// Functions/Drawing/F_VN_DrawMatchesExp

	{attribute 'TcIecLibraryType'}
	{attribute 'external_name' := 'F_VN_DrawMatchesExp_GUID_C69E0A3C_7312_D2B7_BD5B_52E833304808'}
	(* Draws the keypoints and matches for visualization purpose. (expert function) *)
	FUNCTION F_VN_DrawMatchesExp : HRESULT
	VAR_INPUT
		ipSrcImage1	:	ITcVnImage;	(* Source image 1 (elements of type USINT) *)
		ipKeyPoints1	:	ITcVnContainer;	(* Container with the keypoints 1 (ContainerType_Vector_TcVnKeyPoint) *)
		ipSrcImage2	:	ITcVnImage;	(* Source image 2 (elements of type USINT, must have the same number of channels as ipSrcImage1) *)
		ipKeyPoints2	:	ITcVnContainer;	(* Container with the keypoints 2 (ContainerType_Vector_TcVnKeyPoint) *)
		ipMatches1To2	:	ITcVnContainer;	(* Container with the descriptor matches (ContainerType_Vector_TcVnDMatch) *)
		ipDestImage	:	REFERENCE TO ITcVnImage;	(* Destination image (An appropriate color image will be created if required.) *)
	END_VAR
	VAR_IN_OUT
		aMatchColor	:	TcVnVector4_LREAL;	(* Color to draw the matches (for {-1, -1, -1, -1}, a random color is chosen for each point and line) *)
		aSingleColor	:	TcVnVector4_LREAL;	(* Color to draw the single keypoints (for {-1, -1, -1, -1}, a random color is chosen for each point) *)
	END_VAR
	VAR_INPUT
		ipMatchesMask	:	ITcVnContainer;	(* Mask to select the matches to be drawn (ContainerType_Vector_SINT; Set to 0 if all matches should be drawn.) *)
		eFlags	:	ETcVnDrawMatchesFlags;	(* A combination of flags to support overdrawing an existing destination image and/or drawing additional (Rich-)Keypoint information (size and orientation) and/or skipping single keypoints *)
		hrPrev	:	HRESULT;	(* HRESULT indicating the result of previous operations (If SUCCEEDED(hrPrev) equals false, no operation is executed.) *)
	END_VAR

END_FUNCTION

// Functions/Drawing/F_VN_DrawOrientation

	{attribute 'TcIecLibraryType'}
	{attribute 'external_name' := 'F_VN_DrawOrientation_GUID_8C5CCEF9_05D8_D749_BE94_0462EB58FE1E'}
	(* Draw the main axis of a set of points/contour based on a rotated rectangle. *)
	FUNCTION F_VN_DrawOrientation : HRESULT
	VAR_IN_OUT
		stOrientation	:	TcVnRotatedRectangle;	(* Rotated rectangle, containig center of mass, lenghts of axes, and rotation angle in clockwise direction *)
	END_VAR
	VAR_INPUT
		ipDestImage	:	ITcVnImage;	(* Destination image *)
	END_VAR
	VAR_IN_OUT
		aColorMainAxis	:	TcVnVector4_LREAL;	(* Color of the major axis *)
	END_VAR
	VAR_INPUT
		nThickness	:	DINT;	(* Line thickness *)
		hrPrev	:	HRESULT;	(* HRESULT indicating the result of previous operations (If SUCCEEDED(hrPrev) equals false, no operation is executed.) *)
	END_VAR

END_FUNCTION

// Functions/Drawing/F_VN_DrawOrientationExp

	{attribute 'TcIecLibraryType'}
	{attribute 'external_name' := 'F_VN_DrawOrientationExp_GUID_696CB60D_07A4_DDA6_8A99_EB0492A244F0'}
	(* Draw the main axis, the horizontal axis and the angle of a set of points/contour based on a rotated rectangle. (expert function) *)
	FUNCTION F_VN_DrawOrientationExp : HRESULT
	VAR_IN_OUT
		stOrientation	:	TcVnRotatedRectangle;	(* Rotated rectangle, containig center of mass, lenghts of axes, and rotation angle in clockwise direction *)
	END_VAR
	VAR_INPUT
		ipDestImage	:	ITcVnImage;	(* Destination image *)
	END_VAR
	VAR_IN_OUT
		aColorMainAxis	:	TcVnVector4_LREAL;	(* Color of the major axis *)
	END_VAR
	VAR_INPUT
		nThickness	:	DINT;	(* Line thickness *)
	END_VAR
	VAR_IN_OUT
		aColorHorizontalAxis	:	TcVnVector4_LREAL;	(* Color of the horizontal axis *)
	END_VAR
	VAR_INPUT
		fFontScale	:	LREAL;	(* Scaling factor for the text *)
		hrPrev	:	HRESULT;	(* HRESULT indicating the result of previous operations (If SUCCEEDED(hrPrev) equals false, no operation is executed.) *)
	END_VAR

END_FUNCTION

// Functions/Drawing/F_VN_DrawPoint

	{attribute 'TcIecLibraryType'}
	{attribute 'external_name' := 'F_VN_DrawPoint_GUID_EB197B9A_8498_D424_9F64_30D926D7A450'}
	(* Draws a point. *)
	FUNCTION F_VN_DrawPoint : HRESULT
	VAR_INPUT
		nX	:	UDINT;	(* x coordinate of the point *)
		nY	:	UDINT;	(* y coordinate of the point *)
		ipDestImage	:	ITcVnImage;	(* Destination image *)
		eShape	:	ETcVnDrawShape;	(* Point shape *)
	END_VAR
	VAR_IN_OUT
		aColor	:	TcVnVector4_LREAL;	(* Color (for {-1, -1, -1, -1}, a random color is chosen) *)
	END_VAR
	VAR_INPUT
		hrPrev	:	HRESULT;	(* HRESULT indicating the result of previous operations (If SUCCEEDED(hrPrev) equals false, no operation is executed.) *)
	END_VAR

END_FUNCTION

// Functions/Drawing/F_VN_DrawPointExp

	{attribute 'TcIecLibraryType'}
	{attribute 'external_name' := 'F_VN_DrawPointExp_GUID_0CB1EFC6_EA71_DD9E_A07B_08DD7C0269E3'}
	(* Draw a point. (expert function) *)
	FUNCTION F_VN_DrawPointExp : HRESULT
	VAR_INPUT
		nX	:	UDINT;	(* x coordinate of the point *)
		nY	:	UDINT;	(* y coordinate of the point *)
		ipDestImage	:	ITcVnImage;	(* Destination image *)
		eShape	:	ETcVnDrawShape;	(* Point shape *)
	END_VAR
	VAR_IN_OUT
		aColor	:	TcVnVector4_LREAL;	(* Color (for {-1, -1, -1, -1}, a random color is chosen) *)
	END_VAR
	VAR_INPUT
		nSize	:	UDINT;	(* Size of the shape (half width) *)
		nThickness	:	DINT;	(* Line thickness (if negative, the shape is filled if it is closed) *)
		eLineType	:	ETcVnLineType;	(* Line type *)
		hrPrev	:	HRESULT;	(* HRESULT indicating the result of previous operations (If SUCCEEDED(hrPrev) equals false, no operation is executed.) *)
	END_VAR

END_FUNCTION

// Functions/Drawing/F_VN_DrawPoints

	{attribute 'TcIecLibraryType'}
	{attribute 'external_name' := 'F_VN_DrawPoints_GUID_E6C839DF_E6AE_DD7C_B6D1_DE7AB7EFA551'}
	(* Draw a collection of points. *)
	FUNCTION F_VN_DrawPoints : HRESULT
	VAR_INPUT
		ipPoints	:	ITcVnContainer;	(* Container with TcVnPoint2_DINT or TcVnPoint2_REAL elements *)
		ipDestImage	:	ITcVnImage;	(* Destination image *)
		eShape	:	ETcVnDrawShape;	(* Point shape *)
	END_VAR
	VAR_IN_OUT
		aColor	:	TcVnVector4_LREAL;	(* Color (for {-1, -1, -1, -1}, a random color is chosen for each point) *)
	END_VAR
	VAR_INPUT
		hrPrev	:	HRESULT;	(* HRESULT indicating the result of previous operations (If SUCCEEDED(hrPrev) equals false, no operation is executed.) *)
	END_VAR

END_FUNCTION

// Functions/Drawing/F_VN_DrawPointsExp

	{attribute 'TcIecLibraryType'}
	{attribute 'external_name' := 'F_VN_DrawPointsExp_GUID_34B2960B_E925_DF02_A623_3F9677F5FB98'}
	(* Draw a collection of points. (expert function) *)
	FUNCTION F_VN_DrawPointsExp : HRESULT
	VAR_INPUT
		ipPoints	:	ITcVnContainer;	(* Container with TcVnPoint2_DINT or TcVnPoint2_REAL elements *)
		ipDestImage	:	ITcVnImage;	(* Destination image *)
		eShape	:	ETcVnDrawShape;	(* Point shape *)
	END_VAR
	VAR_IN_OUT
		aColor	:	TcVnVector4_LREAL;	(* Color (for {-1, -1, -1, -1}, a random color is chosen for each point) *)
	END_VAR
	VAR_INPUT
		nSize	:	UDINT;	(* Size of the shape (half width) *)
		nThickness	:	DINT;	(* Line thickness (if negative, the shape is filled if it is closed) *)
		eLineType	:	ETcVnLineType;	(* Line type *)
		hrPrev	:	HRESULT;	(* HRESULT indicating the result of previous operations (If SUCCEEDED(hrPrev) equals false, no operation is executed.) *)
	END_VAR

END_FUNCTION

// Functions/Drawing/F_VN_DrawPolygon

	{attribute 'TcIecLibraryType'}
	{attribute 'external_name' := 'F_VN_DrawPolygon_GUID_2AC3D600_E474_DEFB_A3DB_E972A97945F6'}
	(* Draw a pologon using collection of points. *)
	FUNCTION F_VN_DrawPolygon : HRESULT
	VAR_INPUT
		ipPoints	:	ITcVnContainer;	(* Container with TcVnPoint2_DINT, TcVnPoint2_REAL, or TcVnPoint2_LREAL elements *)
		ipDestImage	:	ITcVnImage;	(* Destination image *)
	END_VAR
	VAR_IN_OUT
		aColor	:	TcVnVector4_LREAL;	(* Color *)
	END_VAR
	VAR_INPUT
		nThickness	:	DINT;	(* Line thickness (if negative, the polygon is filled) *)
		hrPrev	:	HRESULT;	(* HRESULT indicating the result of previous operations (If SUCCEEDED(hrPrev) equals false, no operation is executed.) *)
	END_VAR

END_FUNCTION

// Functions/Drawing/F_VN_DrawPolygonExp

	{attribute 'TcIecLibraryType'}
	{attribute 'external_name' := 'F_VN_DrawPolygonExp_GUID_D79A9437_66CC_D2F2_AC2B_AABA5EDF4A83'}
	(* Draw a pologon using collection of points. (expert function) *)
	FUNCTION F_VN_DrawPolygonExp : HRESULT
	VAR_INPUT
		ipPoints	:	ITcVnContainer;	(* Container with TcVnPoint2_DINT, TcVnPoint2_REAL, or TcVnPoint2_LREAL elements *)
		ipDestImage	:	ITcVnImage;	(* Destination image *)
	END_VAR
	VAR_IN_OUT
		aColor	:	TcVnVector4_LREAL;	(* Color *)
	END_VAR
	VAR_INPUT
		nThickness	:	DINT;	(* Line thickness (if negative, the shape is filled) *)
		bIsClosed	:	BOOL;	(* If it is true, the function draws a line from the last point to the first point to close the polygon. *)
		eLineType	:	ETcVnLineType;	(* Line type *)
		nShift	:	UDINT;	(* Fractional bits of the coordinates (bit shift) *)
		hrPrev	:	HRESULT;	(* HRESULT indicating the result of previous operations (If SUCCEEDED(hrPrev) equals false, no operation is executed.) *)
	END_VAR

END_FUNCTION

// Functions/Drawing/F_VN_DrawRectangle

	{attribute 'TcIecLibraryType'}
	{attribute 'external_name' := 'F_VN_DrawRectangle_GUID_CA7621FD_AAA8_DD79_BAA6_54BF18EEF247'}
	(* Draw a rectangle. *)
	FUNCTION F_VN_DrawRectangle : HRESULT
	VAR_INPUT
		nTopLeftX	:	UDINT;	(* x coordinate of the top left corner *)
		nTopLeftY	:	UDINT;	(* y coordinate of the top left corner *)
		nBottomRightX	:	UDINT;	(* x coordinate of the bottom right corner *)
		nBottomRightY	:	UDINT;	(* y coordinate of the bottom right corner *)
		ipDestImage	:	ITcVnImage;	(* Destination image *)
	END_VAR
	VAR_IN_OUT
		aColor	:	TcVnVector4_LREAL;	(* Color *)
	END_VAR
	VAR_INPUT
		nThickness	:	DINT;	(* Line thickness (if negative, the rectangle is filled) *)
		hrPrev	:	HRESULT;	(* HRESULT indicating the result of previous operations (If SUCCEEDED(hrPrev) equals false, no operation is executed.) *)
	END_VAR

END_FUNCTION

// Functions/Drawing/F_VN_DrawRectangle_TcVnRectangle_DINT

	{attribute 'TcIecLibraryType'}
	{attribute 'external_name' := 'F_VN_DrawRectangle_TcVnRectangle_DINT_GUID_35950137_42A1_DD6B_8040_5531524BF69E'}
	(* Draw a rectangle. *)
	FUNCTION F_VN_DrawRectangle_TcVnRectangle_DINT : HRESULT
	VAR_IN_OUT
		stRectangle	:	TcVnRectangle_DINT;	(* Rectangle to be drawn *)
	END_VAR
	VAR_INPUT
		ipDestImage	:	ITcVnImage;	(* Destination image *)
	END_VAR
	VAR_IN_OUT
		aColor	:	TcVnVector4_LREAL;	(* Color *)
	END_VAR
	VAR_INPUT
		nThickness	:	DINT;	(* Line thickness (if negative, the rectangle is filled) *)
		hrPrev	:	HRESULT;	(* HRESULT indicating the result of previous operations (If SUCCEEDED(hrPrev) equals false, no operation is executed.) *)
	END_VAR

END_FUNCTION

// Functions/Drawing/F_VN_DrawRectangle_TcVnRectangle_UDINT

	{attribute 'TcIecLibraryType'}
	{attribute 'external_name' := 'F_VN_DrawRectangle_TcVnRectangle_UDINT_GUID_4B7204C8_DED8_DFCB_8469_BEF3FFA8576B'}
	(* Draw a rectangle. *)
	FUNCTION F_VN_DrawRectangle_TcVnRectangle_UDINT : HRESULT
	VAR_IN_OUT
		stRectangle	:	TcVnRectangle_UDINT;	(* Rectangle to be drawn *)
	END_VAR
	VAR_INPUT
		ipDestImage	:	ITcVnImage;	(* Destination image *)
	END_VAR
	VAR_IN_OUT
		aColor	:	TcVnVector4_LREAL;	(* Color *)
	END_VAR
	VAR_INPUT
		nThickness	:	DINT;	(* Line thickness (if negative, the rectangle is filled) *)
		hrPrev	:	HRESULT;	(* HRESULT indicating the result of previous operations (If SUCCEEDED(hrPrev) equals false, no operation is executed.) *)
	END_VAR

END_FUNCTION

// Functions/Drawing/F_VN_DrawRotatedRectangle

	{attribute 'TcIecLibraryType'}
	{attribute 'external_name' := 'F_VN_DrawRotatedRectangle_GUID_E91FE6CA_6FE6_D9DD_B4B2_DB4AEAF725E4'}
	(* Draw a rectangle. *)
	FUNCTION F_VN_DrawRotatedRectangle : HRESULT
	VAR_IN_OUT
		stRectangle	:	TcVnRotatedRectangle;	(* Rectangle to be drawn (rotation angle in degrees) *)
	END_VAR
	VAR_INPUT
		ipDestImage	:	ITcVnImage;	(* Destination image *)
	END_VAR
	VAR_IN_OUT
		aColor	:	TcVnVector4_LREAL;	(* Color *)
	END_VAR
	VAR_INPUT
		nThickness	:	DINT;	(* Line thickness (if negative, the rectangle is filled) *)
		hrPrev	:	HRESULT;	(* HRESULT indicating the result of previous operations (If SUCCEEDED(hrPrev) equals false, no operation is executed.) *)
	END_VAR

END_FUNCTION

// Functions/Drawing/F_VN_DrawRotatedRectangleExp

	{attribute 'TcIecLibraryType'}
	{attribute 'external_name' := 'F_VN_DrawRotatedRectangleExp_GUID_FE06CB4F_97F7_D420_BF0D_F8C392244530'}
	(* Draw a rectangle. (expert function) *)
	FUNCTION F_VN_DrawRotatedRectangleExp : HRESULT
	VAR_IN_OUT
		stRectangle	:	TcVnRotatedRectangle;	(* Rectangle to be drawn (rotation angle in degrees) *)
	END_VAR
	VAR_INPUT
		ipDestImage	:	ITcVnImage;	(* Destination image *)
	END_VAR
	VAR_IN_OUT
		aColor	:	TcVnVector4_LREAL;	(* Color *)
	END_VAR
	VAR_INPUT
		nThickness	:	DINT;	(* Line thickness (if negative, the rectangle is filled) *)
		eLineType	:	ETcVnLineType;	(* Line type *)
		hrPrev	:	HRESULT;	(* HRESULT indicating the result of previous operations (If SUCCEEDED(hrPrev) equals false, no operation is executed.) *)
	END_VAR

END_FUNCTION

// Functions/Drawing/F_VN_FillCircle

	{attribute 'TcIecLibraryType'}
	{attribute 'external_name' := 'F_VN_FillCircle_GUID_57F72791_EAC2_DD4D_87CB_053D8258EE82'}
	(* Paint a filled circle. *)
	FUNCTION F_VN_FillCircle : HRESULT
	VAR_INPUT
		nCenterX	:	UDINT;	(* x coordinate of the center *)
		nCenterY	:	UDINT;	(* y coordinate of the center *)
		nRadius	:	UDINT;	(* Radius *)
		ipDestImage	:	ITcVnImage;	(* Destination image *)
	END_VAR
	VAR_IN_OUT
		aColor	:	TcVnVector4_LREAL;	(* Color *)
	END_VAR
	VAR_INPUT
		hrPrev	:	HRESULT;	(* HRESULT indicating the result of previous operations (If SUCCEEDED(hrPrev) equals false, no operation is executed.) *)
	END_VAR

END_FUNCTION

// Functions/Drawing/F_VN_FillContours

	{attribute 'TcIecLibraryType'}
	{attribute 'external_name' := 'F_VN_FillContours_GUID_9A17D4B9_08AB_D368_B51D_AE757CA4E5B1'}
	(* Paint a single point set or multiple point sets that are interpreted as contours. *)
	FUNCTION F_VN_FillContours : HRESULT
	VAR_INPUT
		ipContours	:	ITcVnContainer;	(* Single contour (ContainerType_Vector_TcVnPoint2_DINT) or multiple contours (ContainerType_Vector_Vector_TcVnPoint2_DINT) *)
		nContourIndex	:	DINT;	(* Index of a specific contour to be drawn (if negative, all contours within the container are drawn) *)
		ipDestImage	:	ITcVnImage;	(* Destination image *)
	END_VAR
	VAR_IN_OUT
		aColor	:	TcVnVector4_LREAL;	(* Color *)
	END_VAR
	VAR_INPUT
		hrPrev	:	HRESULT;	(* HRESULT indicating the result of previous operations (If SUCCEEDED(hrPrev) equals false, no operation is executed.) *)
	END_VAR

END_FUNCTION

// Functions/Drawing/F_VN_FillEllipse

	{attribute 'TcIecLibraryType'}
	{attribute 'external_name' := 'F_VN_FillEllipse_GUID_5CD99C65_85B9_D8C2_BE64_A5A4252AB0BB'}
	(* Paint a filled ellipse. *)
	FUNCTION F_VN_FillEllipse : HRESULT
	VAR_IN_OUT
		stEllipse	:	TcVnRotatedRectangle;	(* Ellipse to be painted (rotation angle in degrees) *)
	END_VAR
	VAR_INPUT
		ipDestImage	:	ITcVnImage;	(* Destination image *)
	END_VAR
	VAR_IN_OUT
		aColor	:	TcVnVector4_LREAL;	(* Color *)
	END_VAR
	VAR_INPUT
		hrPrev	:	HRESULT;	(* HRESULT indicating the result of previous operations (If SUCCEEDED(hrPrev) equals false, no operation is executed.) *)
	END_VAR

END_FUNCTION

// Functions/Drawing/F_VN_FillPolygon

	{attribute 'TcIecLibraryType'}
	{attribute 'external_name' := 'F_VN_FillPolygon_GUID_25CBE1F6_0702_D828_A491_380DC4B9D8A2'}
	(* Paint a filled pologon using a set of points. *)
	FUNCTION F_VN_FillPolygon : HRESULT
	VAR_INPUT
		ipPoints	:	ITcVnContainer;	(* Container with TcVnPoint2_DINT, TcVnPoint2_REAL, or TcVnPoint2_LREAL elements *)
		ipDestImage	:	ITcVnImage;	(* Destination image *)
	END_VAR
	VAR_IN_OUT
		aColor	:	TcVnVector4_LREAL;	(* Color *)
	END_VAR
	VAR_INPUT
		hrPrev	:	HRESULT;	(* HRESULT indicating the result of previous operations (If SUCCEEDED(hrPrev) equals false, no operation is executed.) *)
	END_VAR

END_FUNCTION

// Functions/Drawing/F_VN_FillRectangle

	{attribute 'TcIecLibraryType'}
	{attribute 'external_name' := 'F_VN_FillRectangle_GUID_B6F6404B_5305_DD2F_82D7_B60633C88882'}
	(* Paint a filled rectangle. *)
	FUNCTION F_VN_FillRectangle : HRESULT
	VAR_INPUT
		nTopLeftX	:	UDINT;	(* x coordinate of the top left corner *)
		nTopLeftY	:	UDINT;	(* y coordinate of the top left corner *)
		nBottomRightX	:	UDINT;	(* x coordinate of the bottom right corner *)
		nBottomRightY	:	UDINT;	(* y coordinate of the bottom right corner *)
		ipDestImage	:	ITcVnImage;	(* Destination image *)
	END_VAR
	VAR_IN_OUT
		aColor	:	TcVnVector4_LREAL;	(* Color *)
	END_VAR
	VAR_INPUT
		hrPrev	:	HRESULT;	(* HRESULT indicating the result of previous operations (If SUCCEEDED(hrPrev) equals false, no operation is executed.) *)
	END_VAR

END_FUNCTION

// Functions/Drawing/F_VN_FillRotatedRectangle

	{attribute 'TcIecLibraryType'}
	{attribute 'external_name' := 'F_VN_FillRotatedRectangle_GUID_051B9FAB_5B48_DFCC_BEE4_115436A91595'}
	(* Paint a filled rectangle. *)
	FUNCTION F_VN_FillRotatedRectangle : HRESULT
	VAR_IN_OUT
		stRectangle	:	TcVnRotatedRectangle;	(* Rectangle to be painted (rotation angle in degrees) *)
	END_VAR
	VAR_INPUT
		ipDestImage	:	ITcVnImage;	(* Destination image *)
	END_VAR
	VAR_IN_OUT
		aColor	:	TcVnVector4_LREAL;	(* Color *)
	END_VAR
	VAR_INPUT
		hrPrev	:	HRESULT;	(* HRESULT indicating the result of previous operations (If SUCCEEDED(hrPrev) equals false, no operation is executed.) *)
	END_VAR

END_FUNCTION

// Functions/Drawing/F_VN_PlotIntensityProfile

	{attribute 'TcIecLibraryType'}
	{attribute 'external_name' := 'F_VN_PlotIntensityProfile_GUID_B2A04906_DDBE_D38C_A697_F571DC74A928'}
	(* Plots the pixel intensity profile along a line segment in an image. *)
	FUNCTION F_VN_PlotIntensityProfile : HRESULT
	VAR_INPUT
		ipSrcImage	:	ITcVnImage;	(* Source image (USINT, 1 channel) *)
		ipDestImage	:	REFERENCE TO ITcVnImage;	(* Destination image (USINT, 1 channel. x: position, y: intensity, origin: bottom left. An appropriate destination image will be created if required.) *)
	END_VAR
	VAR_IN_OUT
		aStartPoint	:	TcVnPoint2_REAL;	(* Start point of the line segment *)
		aEndPoint	:	TcVnPoint2_REAL;	(* End point of the line segment *)
	END_VAR
	VAR_INPUT
		hrPrev	:	HRESULT;	(* HRESULT indicating the result of previous operations (If SUCCEEDED(hrPrev) equals false, no operation is executed.) *)
	END_VAR

END_FUNCTION

// Functions/Drawing/F_VN_PlotIntensityProfileExp

	{attribute 'TcIecLibraryType'}
	{attribute 'external_name' := 'F_VN_PlotIntensityProfileExp_GUID_18DC275F_A530_D420_B515_3BF70FC6163A'}
	(* Plots the pixel intensity profile along a line segment in an image. (expert function) *)
	FUNCTION F_VN_PlotIntensityProfileExp : HRESULT
	VAR_INPUT
		ipSrcImage	:	ITcVnImage;	(* Source image (USINT, 1 channel) *)
		ipDestImage	:	REFERENCE TO ITcVnImage;	(* Destination image (USINT, 1 channel. x: position, y: intensity, origin: bottom left. An appropriate destination image will be created if required.) *)
	END_VAR
	VAR_IN_OUT
		aStartPoint	:	TcVnPoint2_REAL;	(* Start point of the line segment *)
		aEndPoint	:	TcVnPoint2_REAL;	(* End point of the line segment *)
		aBackgroundColor	:	TcVnVector4_LREAL;	(* Background color *)
		aLineColor	:	TcVnVector4_LREAL;	(* Line color *)
		aGridColor	:	TcVnVector4_LREAL;	(* Grid color *)
	END_VAR
	VAR_INPUT
		nScaleX	:	DINT;	(* Scale in x direction (ipDestImage will have a width of nScaleX * (ipSrcImage width - 1) + 1) *)
		nScaleY	:	DINT;	(* Scale in y direction (ipDestImage will have a height of nScaleY * 255 + 1) *)
		nThickness	:	DINT;	(* Line thickness *)
		nDestChannels	:	DINT;	(* ipDestImage channels (1 or 3) *)
		hrPrev	:	HRESULT;	(* HRESULT indicating the result of previous operations (If SUCCEEDED(hrPrev) equals false, no operation is executed.) *)
	END_VAR

END_FUNCTION

// Functions/Drawing/F_VN_PutLabel

	{attribute 'TcIecLibraryType'}
	{attribute 'external_name' := 'F_VN_PutLabel_GUID_AC21311A_53C7_DC28_BB97_DE22D5467497'}
	(* Write a label (black text on white background) into an image. *)
	FUNCTION F_VN_PutLabel : HRESULT
	VAR_IN_OUT CONSTANT
		sText	:	STRING;	(* Text *)
	END_VAR
	VAR_INPUT
		ipDestImage	:	ITcVnImage;	(* Destination image *)
		nX	:	UDINT;	(* x coordinate (bottom left) *)
		nY	:	UDINT;	(* y coordinate (bottom left) *)
		fFontScale	:	LREAL;	(* Scaling factor *)
		hrPrev	:	HRESULT;	(* HRESULT indicating the result of previous operations (If SUCCEEDED(hrPrev) equals false, no operation is executed.) *)
	END_VAR

END_FUNCTION

// Functions/Drawing/F_VN_PutLabelExp

	{attribute 'TcIecLibraryType'}
	{attribute 'external_name' := 'F_VN_PutLabelExp_GUID_22D551B9_953C_DDA8_9D1A_8B55704272D4'}
	(* Write a label (text on unified background) into an image. (expert function) *)
	FUNCTION F_VN_PutLabelExp : HRESULT
	VAR_IN_OUT CONSTANT
		sText	:	STRING;	(* Text *)
	END_VAR
	VAR_INPUT
		ipDestImage	:	ITcVnImage;	(* Destination image *)
		nX	:	UDINT;	(* x coordinate (bottom left) *)
		nY	:	UDINT;	(* y coordinate (bottom left) *)
		fFontScale	:	LREAL;	(* Scaling factor *)
		nThickness	:	UDINT;	(* Line thickness *)
		eFontType	:	ETcVnFontType;	(* Font type *)
	END_VAR
	VAR_IN_OUT
		aFontColor	:	TcVnVector4_LREAL;	(* Font color *)
		aBackgroundColor	:	TcVnVector4_LREAL;	(* Background color *)
	END_VAR
	VAR_INPUT
		eLineType	:	ETcVnLineType;	(* Line type *)
		hrPrev	:	HRESULT;	(* HRESULT indicating the result of previous operations (If SUCCEEDED(hrPrev) equals false, no operation is executed.) *)
	END_VAR

END_FUNCTION

// Functions/Drawing/F_VN_PutText

	{attribute 'TcIecLibraryType'}
	{attribute 'external_name' := 'F_VN_PutText_GUID_8A847AF0_9C61_D376_BA49_31E7BD216F97'}
	(* Write text into an image. *)
	FUNCTION F_VN_PutText : HRESULT
	VAR_IN_OUT CONSTANT
		sText	:	STRING;	(* Text *)
	END_VAR
	VAR_INPUT
		ipDestImage	:	ITcVnImage;	(* Destination image *)
		nX	:	UDINT;	(* x coordinate (bottom left) *)
		nY	:	UDINT;	(* y coordinate (bottom left) *)
		eFontType	:	ETcVnFontType;	(* Font type *)
		fFontScale	:	LREAL;	(* Scaling factor *)
	END_VAR
	VAR_IN_OUT
		aColor	:	TcVnVector4_LREAL;	(* Text color *)
	END_VAR
	VAR_INPUT
		hrPrev	:	HRESULT;	(* HRESULT indicating the result of previous operations (If SUCCEEDED(hrPrev) equals false, no operation is executed.) *)
	END_VAR

END_FUNCTION

// Functions/Drawing/F_VN_PutTextExp

	{attribute 'TcIecLibraryType'}
	{attribute 'external_name' := 'F_VN_PutTextExp_GUID_D88D1077_FEC3_DDA1_8623_3D379A0CC9BD'}
	(* Write text into an image. (expert function) *)
	FUNCTION F_VN_PutTextExp : HRESULT
	VAR_IN_OUT CONSTANT
		sText	:	STRING;	(* Text *)
	END_VAR
	VAR_INPUT
		ipDestImage	:	ITcVnImage;	(* Destination image *)
		nX	:	UDINT;	(* x coordinate (bottom left) *)
		nY	:	UDINT;	(* y coordinate (bottom left) *)
		eFontType	:	ETcVnFontType;	(* Font type *)
		fFontScale	:	LREAL;	(* Scaling factor *)
	END_VAR
	VAR_IN_OUT
		aColor	:	TcVnVector4_LREAL;	(* Text color *)
	END_VAR
	VAR_INPUT
		nThickness	:	DINT;	(* Line thickness *)
		eLineType	:	ETcVnLineType;	(* Line type *)
		bBottomLeftOrigin	:	BOOL;	(* Sets the image origin to the bottom left corner, if true *)
		hrPrev	:	HRESULT;	(* HRESULT indicating the result of previous operations (If SUCCEEDED(hrPrev) equals false, no operation is executed.) *)
	END_VAR

END_FUNCTION

// Functions/Neural Network/F_VN_ConvertDataLayout

	{attribute 'TcIecLibraryType'}
	{attribute 'external_name' := 'F_VN_ConvertDataLayout_GUID_3995A5A2_8722_D5EC_8314_ABF1AA7937E5'}
	(* Convert a data layout (the arrangement of dimensions in the input data) to another data layout. *)
	FUNCTION F_VN_ConvertDataLayout : HRESULT
	VAR_INPUT
		ipSrcImage	:	ITcVnImage;	(* Source image *)
		ipDestImage	:	REFERENCE TO ITcVnImage;	(* Destination image (An appropriate destination image will be created if required.) *)
		nSrcDataLayout	:	ULINT;	(* Data layout of the source image (Commonly used data layouts are available in the enumeration ETcVnDataLayout. If nSrcDataLayout is set to 0 or TCVN_DL_DEFAULT, the DataLayout will be automatically determined based on the dimension of the ipSrcImage: 0x12 for 2D, 0x123 for 3D, 0x1234 for 4D, and so forth.) *)
		nDestDataLayout	:	ULINT;	(* Required output data layout (Commonly used data layouts are available in the enumeration ETcVnDataLayout. nDestDataLayout must not equal 0 or TCVN_DL_DEFAULT.) *)
		hrPrev	:	HRESULT;	(* HRESULT indicating the result of previous operations (If SUCCEEDED(hrPrev) equals false, no operation is executed.) *)
	END_VAR

END_FUNCTION

// Functions/Neural Network/F_VN_ReshapeImage

	{attribute 'TcIecLibraryType'}
	{attribute 'external_name' := 'F_VN_ReshapeImage_GUID_2BBA238A_D9C8_DF6C_A475_21C0DD3F001A'}
	(* Changes the shape of an ITcVnImage. The total number of elements in the new shape must be equal to the total number of elements in ipSrcImage. *)
	FUNCTION F_VN_ReshapeImage : HRESULT
	VAR_INPUT
		ipSrcImage	:	ITcVnImage;	(* Source image (1 channel) *)
		ipDestImage	:	REFERENCE TO ITcVnImage;	(* Destination image (An appropriate single channel destination image will be created if required.) *)
	END_VAR
	VAR_IN_OUT
		aNewShape	:	TcVnArray33_UDINT;	(* Specifies the shape of ipDestImage. First entry is the number of dimensions (max. 32), followed by the sizes of each dimension. If one dimension is set to zero, its value will be automatically calculated based on the total elements of ipSrcImage (Only one dimension can be set to zero.) *)
	END_VAR
	VAR_INPUT
		hrPrev	:	HRESULT;	(* HRESULT indicating the result of previous operations (If SUCCEEDED(hrPrev) equals false, no operation is executed.) *)
	END_VAR

END_FUNCTION

// Functions/Neural Network/F_VN_Sigmoid

	{attribute 'TcIecLibraryType'}
	{attribute 'external_name' := 'F_VN_Sigmoid_GUID_443EE66B_FF0F_D007_AC8F_462BC3F1F276'}
	(* Apply the standard logistic function 1 / (1 + exp(-x)) element-wise to a single- or multi-channel REAL image. *)
	FUNCTION F_VN_Sigmoid : HRESULT
	VAR_INPUT
		ipSrcImage	:	ITcVnImage;	(* Source image (REAL) *)
		ipDestImage	:	REFERENCE TO ITcVnImage;	(* Destination image (An appropriate destination image will be created if required.) *)
		hrPrev	:	HRESULT;	(* HRESULT indicating the result of previous operations (If SUCCEEDED(hrPrev) equals false, no operation is executed.) *)
	END_VAR

END_FUNCTION

// Functions/Neural Network/F_VN_SigmoidExp

	{attribute 'TcIecLibraryType'}
	{attribute 'external_name' := 'F_VN_SigmoidExp_GUID_B65ACE1F_A3FF_DF19_9C9E_6A823D2620ED'}
	(* Apply the logistic function 1 / (1 + exp(-fSteepness * (x - fShift))) element-wise to a single- or multi-channel REAL image. (expert function) *)
	FUNCTION F_VN_SigmoidExp : HRESULT
	VAR_INPUT
		ipSrcImage	:	ITcVnImage;	(* Source image (REAL) *)
		ipDestImage	:	REFERENCE TO ITcVnImage;	(* Destination image (An appropriate destination image will be created if required.) *)
		fShift	:	REAL;	(* Determines the intensity level around which the logistic function transitions. *)
		fSteepness	:	REAL;	(* Controls the sharpness of the transition. *)
		hrPrev	:	HRESULT;	(* HRESULT indicating the result of previous operations (If SUCCEEDED(hrPrev) equals false, no operation is executed.) *)
	END_VAR

END_FUNCTION

// Functions/Neural Network/F_VN_SoftMax

	{attribute 'TcIecLibraryType'}
	{attribute 'external_name' := 'F_VN_SoftMax_GUID_62A1500E_9919_D189_8BB6_E8BC05C5CB3D'}
	(* Apply softmax function pixel-wise to a single channel REAL image. *)
	FUNCTION F_VN_SoftMax : HRESULT
	VAR_INPUT
		ipSrcImage	:	ITcVnImage;	(* Source image (REAL, 1 channel) *)
		ipDestImage	:	REFERENCE TO ITcVnImage;	(* Destination image (An appropriate single channel destination image will be created if required.) *)
		bFlatten	:	BOOL;	(* If true, the resulting image will be reshaped into a single row. *)
		hrPrev	:	HRESULT;	(* HRESULT indicating the result of previous operations (If SUCCEEDED(hrPrev) equals false, no operation is executed.) *)
	END_VAR

END_FUNCTION

// Functions/Neural Network/F_VN_NonMaxSuppression

	{attribute 'TcIecLibraryType'}
	{attribute 'external_name' := 'F_VN_NonMaxSuppression_GUID_DDD612EA_2DB6_D0A1_AA79_316039076A43'}
	(* Perform non-maximum suppression on given bounding boxes and corresponding scores. *)
	FUNCTION F_VN_NonMaxSuppression : HRESULT
	VAR_INPUT
		ipBoundingBoxes	:	ITcVnContainer;	(* Container of bounding boxes to apply the non maximum supresion (ContainerType_Vector_TcVnRectangle_DINT) *)
		ipScores	:	ITcVnContainer;	(* Container of coreeponding score for each bounding box (ContainerType_Vector_REAL) *)
		ipDestIndcies	:	REFERENCE TO ITcVnContainer;	(* Container of the kept indcies after apply the non maximum suppression (ContainerType_Vector_DINT) *)
		fScoreThreshold	:	REAL;	(* A threshold [0.0 to 1.0] used to filter the bounding boxes by score *)
		fOverlapThreshold	:	REAL;	(* A threshold [0.0 to 1.0] that determines the minimum degree of intersection over union (IoU) required for bounding boxes to be considered overlapping *)
		hrPrev	:	HRESULT;	(* HRESULT indicating the result of previous operations (If SUCCEEDED(hrPrev) equals false, no operation is executed.) *)
	END_VAR

END_FUNCTION

// Functions/Neural Network/F_VN_NonMaxSuppressionExp

	{attribute 'TcIecLibraryType'}
	{attribute 'external_name' := 'F_VN_NonMaxSuppressionExp_GUID_254301EF_EB55_D9F0_8663_C0A211C69477'}
	(* Perform non-maximum suppression on given bounding boxes and corresponding scores. (expert function) *)
	FUNCTION F_VN_NonMaxSuppressionExp : HRESULT
	VAR_INPUT
		ipBoundingBoxes	:	ITcVnContainer;	(* Container of bounding boxes to apply the non maximum supresion (ContainerType_Vector_TcVnRectangle_DINT) *)
		ipScores	:	ITcVnContainer;	(* Container of coreeponding score for each bounding box (ContainerType_Vector_REAL) *)
		ipDestIndcies	:	REFERENCE TO ITcVnContainer;	(* Container of the kept indcies after apply the non maximum suppression (ContainerType_Vector_DINT) *)
		fScoreThreshold	:	REAL;	(* A threshold [0.0 to 1.0] used to filter the bounding boxes by score *)
		fOverlapThreshold	:	REAL;	(* A threshold [0.0 to 1.0] that determines the minimum degree of intersection over union (IoU) required for bounding boxes to be considered overlapping *)
		ipClassIndcies	:	ITcVnContainer;	(* Container of corresponding set of class indcies (ContainerType_Vector_DINT) *)
		fEta	:	REAL;	(* An adjustable threshold [0.0 to 1.0] used to dynamically reduce the overlap threshold during processing. Setting it to 1 maintains a constant value for the overlap threshold *)
		nTopK	:	DINT;	(* The maximum number of bounding boxes with the highest scores to undergo the suppression algorithm (must be >= 0). Setting it to zero applies the algorithm to all bounding boxes *)
		hrPrev	:	HRESULT;	(* HRESULT indicating the result of previous operations (If SUCCEEDED(hrPrev) equals false, no operation is executed.) *)
	END_VAR

END_FUNCTION

// Functions/Neural Network/F_VN_ExecuteNeuralNetwork

	{attribute 'TcIecLibraryType'}
	{attribute 'external_name' := 'F_VN_ExecuteNeuralNetwork_GUID_617005B4_6D6B_DC13_A8ED_07F2C339BFC4'}
	(* Execute a neural network using the provided image as input and provide the output of one output layer. The function doesn't perform any pre-processing or transformation. *)
	FUNCTION F_VN_ExecuteNeuralNetwork : HRESULT
	VAR_INPUT
		ipNeuralNetwork	:	ITcVnNeuralNetwork;	(* Neural network model *)
		ipSrcImage	:	ITcVnImage;	(* Source image (The image layout must be adapted to match the model's expected input format using e.g. F_VN_ConvertDataLayout or F_VN_ReshapeImage functions if necessary.) *)
		ipDestImage	:	REFERENCE TO ITcVnImage;	(* Destination image (An appropriate destination image based on the output layer is created. To process the destination image, use e.g. F_VN_ConvertDataLayout or F_VN_ReshapeImage if necessary. *)
		hrPrev	:	HRESULT;	(* HRESULT indicating the result of previous operations (If SUCCEEDED(hrPrev) equals false, no operation is executed.) *)
	END_VAR

END_FUNCTION

// Functions/Neural Network/F_VN_ExecuteNeuralNetwork_MI

	{attribute 'TcIecLibraryType'}
	{attribute 'external_name' := 'F_VN_ExecuteNeuralNetwork_MI_GUID_B9E22B87_BE93_D412_867E_51918F035B7B'}
	(* Execute a neural network with multiple inputs (MI) using the provided images. Ensure all model input names are listed in sInputNames and that the images and names are in the same order. The result of one output layer is returned. The function doesn't perform any pre-processing or transformation. *)
	FUNCTION F_VN_ExecuteNeuralNetwork_MI : HRESULT
	VAR_INPUT
		ipNeuralNetwork	:	ITcVnNeuralNetwork;	(* Neural network model *)
		pSrcImages	:	PVOID;	(* Pointer to an array of source input images *)
		nSrcArraySize	:	UINT;	(* The size of the array referenced by pSrcImages. pSrcImages must reference an array with a size equal to the number of model inputs. *)
	END_VAR
	VAR_IN_OUT CONSTANT
		sInputNames	:	STRING;	(* Input names separated by ";" *)
	END_VAR
	VAR_INPUT
		ipDestImage	:	REFERENCE TO ITcVnImage;	(* Destination image (An appropriate destination image based on the output layer is created. To process the destination image, use e.g. F_VN_ConvertDataLayout or F_VN_ReshapeImage if necessary. *)
		hrPrev	:	HRESULT;	(* HRESULT indicating the result of previous operations (If SUCCEEDED(hrPrev) equals false, no operation is executed.) *)
	END_VAR

END_FUNCTION

// Functions/Neural Network/F_VN_ExecuteNeuralNetwork_MultiLayerOutput

	{attribute 'TcIecLibraryType'}
	{attribute 'external_name' := 'F_VN_ExecuteNeuralNetwork_MultiLayerOutput_GUID_C5CF9BE3_85FE_D822_8CCE_67AE7CEBB5FD'}
	(* This function is deprecated, please use F_VN_ExecuteNeuralNetwork_MO. Execute a neural network using the provided image as input and provide the output of the specified output layers. The function doesn't perform any pre-processing or transformation. *)
	FUNCTION F_VN_ExecuteNeuralNetwork_MultiLayerOutput : HRESULT
	VAR_INPUT
		ipNeuralNetwork	:	ITcVnNeuralNetwork;	(* Neural network model *)
		ipSrcImage	:	ITcVnImage;	(* Source image (The image layout must be adapted to match the model's expected input format using e.g. F_VN_ConvertDataLayout or F_VN_ReshapeImage functions if necessary.) *)
		ipDestImages	:	REFERENCE TO ITcVnContainer;	(* Container of images containing the output from the specified layers. *)
		ipLayerNames	:	ITcVnContainer;	(* Container of layer names whose outputs to be returned (ContainerType_Vector_String_SINT). If set to zero, the outputs of all unconnected output layers will be returned.. *)
		hrPrev	:	HRESULT;	(* HRESULT indicating the result of previous operations (If SUCCEEDED(hrPrev) equals false, no operation is executed.) *)
	END_VAR

END_FUNCTION

// Functions/Neural Network/F_VN_ExecuteNeuralNetwork_MO

	{attribute 'TcIecLibraryType'}
	{attribute 'external_name' := 'F_VN_ExecuteNeuralNetwork_MO_GUID_6AF35397_B5CA_D20E_B2FF_C345DD38CC9E'}
	(* Execute a neural network using the provided image as input and provide the output of the specified output layers. The function doesn't perform any pre-processing or transformation. *)
	FUNCTION F_VN_ExecuteNeuralNetwork_MO : HRESULT
	VAR_INPUT
		ipNeuralNetwork	:	ITcVnNeuralNetwork;	(* Neural network model *)
		ipSrcImage	:	ITcVnImage;	(* Source image (The image layout must be adapted to match the model's expected input format using e.g. F_VN_ConvertDataLayout or F_VN_ReshapeImage functions if necessary.) *)
		ipDestImages	:	REFERENCE TO ITcVnContainer;	(* Container of images containing the output from the specified layers. *)
		ipOutputNames	:	ITcVnContainer;	(* Container of layer names whose outputs to be returned (ContainerType_Vector_String_SINT). If set to zero, the outputs of all unconnected output layers will be returned.. *)
		hrPrev	:	HRESULT;	(* HRESULT indicating the result of previous operations (If SUCCEEDED(hrPrev) equals false, no operation is executed.) *)
	END_VAR

END_FUNCTION

// Functions/Neural Network/F_VN_ExecuteNeuralNetwork_MIMO_String

	{attribute 'TcIecLibraryType'}
	{attribute 'external_name' := 'F_VN_ExecuteNeuralNetwork_MIMO_String_GUID_79262195_4885_D38F_BFB4_852FB2DA88FA'}
	(* Execute a neural network with multiple inputs and multiple outputs (MIMO) using the provided images. Ensure all model input names are listed in sInputNames and that the images and names are in the same order. The result of the specified output layers are returned. The function doesn't perform any pre-processing or transformation. *)
	FUNCTION F_VN_ExecuteNeuralNetwork_MIMO_String : HRESULT
	VAR_INPUT
		ipNeuralNetwork	:	ITcVnNeuralNetwork;	(* Neural network model *)
		pSrcImages	:	PVOID;	(* Pointer to an array of source input images *)
		nSrcArraySize	:	UINT;	(* The size of the array referenced by pSrcImages. pSrcImages must reference an array with a size equal to the number of model inputs. *)
	END_VAR
	VAR_IN_OUT CONSTANT
		sInputNames	:	STRING;	(* Input names separated by ";" *)
	END_VAR
	VAR_INPUT
		ipDestImages	:	REFERENCE TO ITcVnContainer;	(* Container of images containing the output from the specified layers. *)
	END_VAR
	VAR_IN_OUT CONSTANT
		sOutputNames	:	STRING;	(* Names of output layers whose outputs are required separated by ";". If empty, the outputs of all unconnected output layers are provided. *)
	END_VAR
	VAR_INPUT
		hrPrev	:	HRESULT;	(* HRESULT indicating the result of previous operations (If SUCCEEDED(hrPrev) equals false, no operation is executed.) *)
	END_VAR

END_FUNCTION

// Functions/Neural Network/F_VN_ExecuteNeuralNetwork_SingleLayerOutput

	{attribute 'TcIecLibraryType'}
	{attribute 'external_name' := 'F_VN_ExecuteNeuralNetwork_SingleLayerOutput_GUID_1A89F6CC_9C3C_D33C_8988_5490C4182C8C'}
	(* This function is deprecated, please use F_VN_ExecuteNeuralNetwork_SO. Execute a neural network using the provided image as input and provide the output of the specified output layer. The function doesn't perform any pre-processing or transformation. *)
	FUNCTION F_VN_ExecuteNeuralNetwork_SingleLayerOutput : HRESULT
	VAR_INPUT
		ipNeuralNetwork	:	ITcVnNeuralNetwork;	(* Neural network model *)
		ipSrcImage	:	ITcVnImage;	(* Source image (The image layout must be adapted to match the model's expected input format using e.g. F_VN_ConvertDataLayout or F_VN_ReshapeImage functions if necessary.) *)
		ipDestImage	:	REFERENCE TO ITcVnImage;	(* Destination image (An appropriate destination image based on the output layer is created. To process the destination image, use e.g. F_VN_ConvertDataLayout or F_VN_ReshapeImage if necessary. *)
	END_VAR
	VAR_IN_OUT CONSTANT
		sLayerName	:	STRING;	(* Specify the name of the layer for which the output is required. If empty, the output of one output layer is provided. *)
	END_VAR
	VAR_INPUT
		hrPrev	:	HRESULT;	(* HRESULT indicating the result of previous operations (If SUCCEEDED(hrPrev) equals false, no operation is executed.) *)
	END_VAR

END_FUNCTION

// Functions/Neural Network/F_VN_ExecuteNeuralNetwork_SO

	{attribute 'TcIecLibraryType'}
	{attribute 'external_name' := 'F_VN_ExecuteNeuralNetwork_SO_GUID_A81F4078_B42F_D9B3_A6A4_C74C5385CC0D'}
	(* Execute a neural network using the provided image as input and provide the output of the specified output layer. The function doesn't perform any pre-processing or transformation. *)
	FUNCTION F_VN_ExecuteNeuralNetwork_SO : HRESULT
	VAR_INPUT
		ipNeuralNetwork	:	ITcVnNeuralNetwork;	(* Neural network model *)
		ipSrcImage	:	ITcVnImage;	(* Source image (The image layout must be adapted to match the model's expected input format using e.g. F_VN_ConvertDataLayout or F_VN_ReshapeImage functions if necessary.) *)
		ipDestImage	:	REFERENCE TO ITcVnImage;	(* Destination image (An appropriate destination image based on the output layer is created. To process the destination image, use e.g. F_VN_ConvertDataLayout or F_VN_ReshapeImage if necessary. *)
	END_VAR
	VAR_IN_OUT CONSTANT
		sOutputName	:	STRING;	(* Specify the name of the layer for which the output is required. If empty, the output of one output layer is provided. *)
	END_VAR
	VAR_INPUT
		hrPrev	:	HRESULT;	(* HRESULT indicating the result of previous operations (If SUCCEEDED(hrPrev) equals false, no operation is executed.) *)
	END_VAR

END_FUNCTION

// Functions/Neural Network/F_VN_ExecuteNeuralNetwork_MISO

	{attribute 'TcIecLibraryType'}
	{attribute 'external_name' := 'F_VN_ExecuteNeuralNetwork_MISO_GUID_CF6E09EA_1398_D740_AF29_8EF8732EB380'}
	(* Execute a neural network with multiple inputs and single output (MISO) using the provided images. Ensure all model input names are listed in sInputNames and that the images and names are in the same order. The result of the specified output layer is returned. The function doesn't perform any pre-processing or transformation. *)
	FUNCTION F_VN_ExecuteNeuralNetwork_MISO : HRESULT
	VAR_INPUT
		ipNeuralNetwork	:	ITcVnNeuralNetwork;	(* Neural network model *)
		pSrcImages	:	PVOID;	(* Pointer to an array of source input images *)
		nSrcArraySize	:	UINT;	(* The size of the array referenced by pSrcImages. pSrcImages must reference an array with a size equal to the number of model inputs. *)
	END_VAR
	VAR_IN_OUT CONSTANT
		sInputNames	:	STRING;	(* Input names separated by ";" *)
	END_VAR
	VAR_INPUT
		ipDestImage	:	REFERENCE TO ITcVnImage;	(* Destination image (An appropriate destination image based on the output layer is created. To process the destination image, use e.g. F_VN_ConvertDataLayout or F_VN_ReshapeImage if necessary. *)
	END_VAR
	VAR_IN_OUT CONSTANT
		sOutputName	:	STRING;	(* Specify the name of the layer for which the output is required. If empty, the output of one output layer is provided. *)
	END_VAR
	VAR_INPUT
		hrPrev	:	HRESULT;	(* HRESULT indicating the result of previous operations (If SUCCEEDED(hrPrev) equals false, no operation is executed.) *)
	END_VAR

END_FUNCTION

// Functions/Neural Network/F_VN_GetNeuralNetworkLayerNames

	{attribute 'TcIecLibraryType'}
	{attribute 'external_name' := 'F_VN_GetNeuralNetworkLayerNames_GUID_223B1AF8_B72E_D672_874C_ECB2B3909417'}
	(* Get the name of all layers in the neural network model. If the bOnlyOuput flag is set to true, only the unconnected output layer names are returned. *)
	FUNCTION F_VN_GetNeuralNetworkLayerNames : HRESULT
	VAR_INPUT
		ipNeuralNetwork	:	ITcVnNeuralNetwork;	(* Neural network model *)
		ipLayerNames	:	REFERENCE TO ITcVnContainer;	(* Container with the layers names (ContainerType_Vector_String_SINT)  *)
		bOnlyOutputs	:	BOOL;	(* If true, only the unconnected output layer names are returned. *)
		hrPrev	:	HRESULT;	(* HRESULT indicating the result of previous operations (If SUCCEEDED(hrPrev) equals false, no operation is executed.) *)
	END_VAR

END_FUNCTION

// Functions/Neural Network/F_VN_GetNeuralNetworkLayerNamesExp

	{attribute 'TcIecLibraryType'}
	{attribute 'external_name' := 'F_VN_GetNeuralNetworkLayerNamesExp_GUID_63C46346_C412_D41B_A47F_D3FCD28AFEC4'}
	(* Get the name of model layers in the neural network model. (expert function) *)
	FUNCTION F_VN_GetNeuralNetworkLayerNamesExp : HRESULT
	VAR_INPUT
		ipNeuralNetwork	:	ITcVnNeuralNetwork;	(* Neural network model *)
		ipLayerNames	:	REFERENCE TO ITcVnContainer;	(* Container with the layers names (ContainerType_Vector_String_SINT) *)
		eLayerNameType	:	ETcVnLayerNameType;	(* Layer name type *)
		hrPrev	:	HRESULT;	(* HRESULT indicating the result of previous operations (If SUCCEEDED(hrPrev) equals false, no operation is executed.) *)
	END_VAR

END_FUNCTION

// Functions/Neural Network/F_VN_GetNeuralNetworkLayerNamesExp_String

	{attribute 'TcIecLibraryType'}
	{attribute 'external_name' := 'F_VN_GetNeuralNetworkLayerNamesExp_String_GUID_8DEA8301_FECD_D62C_897C_03D1F8825FA6'}
	(* Get the name of model layers in the neural network model. (expert function) *)
	FUNCTION F_VN_GetNeuralNetworkLayerNamesExp_String : HRESULT
	VAR_INPUT
		ipNeuralNetwork	:	ITcVnNeuralNetwork;	(* Neural network model *)
	END_VAR
	VAR_IN_OUT CONSTANT
		sLayerNames	:	STRING;	(* Layer names separated by ";". Make sure to choose a sufficient STRING size! *)
	END_VAR
	VAR_INPUT
		nMaxLength	:	ULINT;	(* Maximum string length to export (including 0 termination). If the container content is longer, the string is cut off at nMaxLength - 1 and 0 termination is appended. In this case, S_FALSE is returned. *)
		eLayerNameType	:	ETcVnLayerNameType;	(* Layer name type *)
		hrPrev	:	HRESULT;	(* HRESULT indicating the result of previous operations (If SUCCEEDED(hrPrev) equals false, no operation is executed.) *)
	END_VAR

END_FUNCTION

// Functions/Neural Network/F_VN_Reduce

	{attribute 'TcIecLibraryType'}
	{attribute 'external_name' := 'F_VN_Reduce_GUID_63B76DDC_463A_D386_80ED_3AA5E84AFF33'}
	(* Reduce ipSrcImage by applying the specified operation across rows/columns to obtain a single row/column/channel with the resulting values. *)
	FUNCTION F_VN_Reduce : HRESULT
	VAR_INPUT
		ipSrcImage	:	ITcVnImage;	(* Source image (USINT or REAL elements, 1 channel) *)
		ipDestImage	:	REFERENCE TO ITcVnImage;	(* Destination image. If ipSrcImage is of type USINT and the reduction type is SUM or AVG, ipDestImage will be of type REAL; otherwise, it retains the same type as ipSrcImage (An appropriate single channel destination image will be created if required.) *)
		nDim	:	DINT;	(* Index along which the ITcVnImage is reduced: 0 reduces the matrix to a single row, 1 reduces it to a single column, and 2 reduces to a single channel *)
		eReduceType	:	ETcVnReduceType;	(* Reduction operation *)
		hrPrev	:	HRESULT;	(* HRESULT indicating the result of previous operations (If SUCCEEDED(hrPrev) equals false, no operation is executed.) *)
	END_VAR

END_FUNCTION

// Functions/Neural Network/F_VN_ReduceArg

	{attribute 'TcIecLibraryType'}
	{attribute 'external_name' := 'F_VN_ReduceArg_GUID_84382ACA_A419_DECD_9B4F_A672F72D29A2'}
	(* Finds indices of max/min elements along provided axis and reduce the ipSrcImage to a single row/column/channel. *)
	FUNCTION F_VN_ReduceArg : HRESULT
	VAR_INPUT
		ipSrcImage	:	ITcVnImage;	(* Source image *)
		ipDestImage	:	REFERENCE TO ITcVnImage;	(* Destination image of type DINT (An appropriate single channel destination image will be created if required.) *)
		nDim	:	DINT;	(* Index along which the ipSrcImage is reduced: 0 reduces the matrix to a single row, 1 reduces it to a single column, and 2 reduces to a single channel *)
		eReduceType	:	DINT;	(* Reduction operation REDUCE_MAX or REDUCE_MIN *)
		hrPrev	:	HRESULT;	(* HRESULT indicating the result of previous operations (If SUCCEEDED(hrPrev) equals false, no operation is executed.) *)
	END_VAR

END_FUNCTION

// Functions/Keypoint Features/F_VN_FilterGoodMatches

	{attribute 'TcIecLibraryType'}
	{attribute 'external_name' := 'F_VN_FilterGoodMatches_GUID_1FA03519_29D9_D86E_9508_65D2DBF759BF'}
	(* Filter the descriptor matches and return only good ones. *)
	FUNCTION F_VN_FilterGoodMatches : HRESULT
	VAR_INPUT
		ipMatches	:	ITcVnContainer;	(* Container with descriptor matches (ContainerType_Vector_TcVnDMatch or ContainerType_Vector_Vector_TcVnDMatch) *)
		ipGoodMatches	:	REFERENCE TO ITcVnContainer;	(* Returns a container with good matches (ContainerType_Vector_TcVnDMatch) *)
		fMaxDist	:	REAL;	(* Maximum allowed descriptor distance (-1 disables this filter criterion) *)
		fMaxKnnRatio	:	REAL;	(* Maximum allowed distance ratio between first and second best match ([0..1], used for knn match results only, -1 disables this filter criterion) *)
		hrPrev	:	HRESULT;	(* HRESULT indicating the result of previous operations (If SUCCEEDED(hrPrev) equals false, no operation is executed.) *)
	END_VAR

END_FUNCTION

// Functions/Keypoint Features/F_VN_FindReferenceKeyPointsInImage

	{attribute 'TcIecLibraryType'}
	{attribute 'external_name' := 'F_VN_FindReferenceKeyPointsInImage_GUID_1EF9B151_0275_DE01_8C96_B760837FB991'}
	(* Searches a reference image, represented by its keypoints and corresponding descriptors, in a given source image. *)
	FUNCTION F_VN_FindReferenceKeyPointsInImage : HRESULT
	VAR_INPUT
		ipSrcKeyPoints	:	ITcVnContainer;	(* KeyPoints of the source image, e.g. (ContainerType_Vector_TcVnKeyPoint) *)
		ipSrcDescriptors	:	ITcVnImage;	(* Descriptors of the source image KeyPoints *)
		ipRefKeyPoints	:	ITcVnContainer;	(* KeyPoints of the reference image, e.g. (ContainerType_Vector_TcVnKeyPoint) *)
		ipRefDescriptors	:	ITcVnImage;	(* Descriptors of the reference image KeyPoints *)
		nRefImageWidth	:	UDINT;	(* Width of the reference image in pixels *)
		nRefImageHeight	:	UDINT;	(* Height of the reference image in pixels *)
		ipEdgePoints	:	REFERENCE TO ITcVnContainer;	(* Returns a container with the 4 edge points of the reference image transformed into the coordinates of the source image (ContainerType_Vector_TcVnPoint2_REAL) *)
		fMaxDist	:	REAL;	(* Maximum allowed descriptor distance (-1 disables this filter criterion) *)
		fMaxKnnRatio	:	REAL;	(* Maximum allowed distance ratio between first and second best match ([0..1], -1 disables this filter criterion) *)
		eNormType	:	ETcVnNormalizationType;	(* Normalization type used for descriptor matching (HAMMING recommended for AKAZE, ORB, and BRISK. HAMMING2 is recommended for ORB if the ORB nBriefPoints parameter is 3 or 4. ) *)
		hrPrev	:	HRESULT;	(* HRESULT indicating the result of previous operations (If SUCCEEDED(hrPrev) equals false, no operation is executed.) *)
	END_VAR
	VAR_OUTPUT
		aPerspectiveTransform	:	TcVnMatrix3x3_LREAL;	(* Returns the perspective transformation matrix, which transforms the reference points to the source points *)
		nNumberOfGoodMatches	:	UDINT;	(* Return the number of good matches *)
		nNumberOfInliers	:	UDINT;	(* Return the number of inlier matches *)
	END_VAR

END_FUNCTION

// Functions/Keypoint Features/F_VN_FindReferenceKeyPointsInImageExp

	{attribute 'TcIecLibraryType'}
	{attribute 'external_name' := 'F_VN_FindReferenceKeyPointsInImageExp_GUID_5A9A4E8E_2880_DEC5_B002_F6B228166183'}
	(* Searches a reference image, represented by its keypoints and corresponding descriptors, in a given source image. (expert function) *)
	FUNCTION F_VN_FindReferenceKeyPointsInImageExp : HRESULT
	VAR_INPUT
		ipSrcKeyPoints	:	ITcVnContainer;	(* KeyPoints of the source image, e.g. (ContainerType_Vector_TcVnKeyPoint) *)
		ipSrcDescriptors	:	ITcVnImage;	(* Descriptors of the source image KeyPoints *)
		ipRefKeyPoints	:	ITcVnContainer;	(* KeyPoints of the reference image (ContainerType_Vector_TcVnKeyPoint) *)
		ipRefDescriptors	:	ITcVnImage;	(* Descriptors of the reference image KeyPoints *)
		nRefImageWidth	:	UDINT;	(* Width of the reference image in pixels *)
		nRefImageHeight	:	UDINT;	(* Height of the reference image in pixels *)
		ipEdgePoints	:	REFERENCE TO ITcVnContainer;	(* Returns a container with the 4 edge points of the reference image transformed into the coordinates of the source image (ContainerType_Vector_TcVnPoint2_REAL) *)
		fMaxDist	:	REAL;	(* Maximum allowed descriptor distance (-1 disables this filter criterion) *)
		fMaxKnnRatio	:	REAL;	(* Maximum allowed distance ratio between first and second best match ([0..1], -1 disables this filter criterion) *)
		eNormType	:	ETcVnNormalizationType;	(* Normalization type used for descriptor matching (HAMMING recommended for AKAZE, ORB, and BRISK. HAMMING2 is recommended for ORB if the ORB nBriefPoints parameter is 3 or 4. ) *)
		eAlgorithm	:	ETcVnEstimationAlgorithm;	(* Estimation algorithm used for computing the perspective transformation between the two point sets *)
		fReprojThreshold	:	LREAL;	(* Maximum allowed reprojection error to treat a point pair as an inlier (only used if eAlgorithm is RANSAC, RHO) *)
		nMaxIterations	:	UDINT;	(* Maximum number of RANSAC iterations *)
		fConfidence	:	LREAL;	(* Confidence (0..1) *)
		ipGoodMatches	:	REFERENCE TO ITcVnContainer;	(* Returns a container with good matches (optional, set to 0 if not required; ContainerType_Vector_TcVnDMatch) *)
		ipInlierMask	:	REFERENCE TO ITcVnContainer;	(* Returns a mask marking the inliers (optional, set to 0 if not required; ContainerType_Vector_SINT; only for RANSAC, LMEDS) *)
		hrPrev	:	HRESULT;	(* HRESULT indicating the result of previous operations (If SUCCEEDED(hrPrev) equals false, no operation is executed.) *)
	END_VAR
	VAR_OUTPUT
		aPerspectiveTransform	:	TcVnMatrix3x3_LREAL;	(* Returns the perspective transformation matrix, which transforms the reference points to the source points  *)
		nNumberOfGoodMatches	:	UDINT;	(* Return the number of good matches *)
		nNumberOfInliers	:	UDINT;	(* Return the number of inlier matches *)
	END_VAR

END_FUNCTION

// Functions/Keypoint Features/F_VN_FindReferenceKeyPointsInImageAKAZE

	{attribute 'TcIecLibraryType'}
	{attribute 'external_name' := 'F_VN_FindReferenceKeyPointsInImageAKAZE_GUID_266D06B3_DFB3_D579_B8B6_F6FF64EFE56F'}
	(* Searches a reference image, represented by its AKAZE keypoints and corresponding descriptors, in a given source image (uses the default TcVnParamsAKAZE parameters). *)
	FUNCTION F_VN_FindReferenceKeyPointsInImageAKAZE : HRESULT
	VAR_INPUT
		ipSrcImage	:	ITcVnImage;	(* Source image *)
		ipRefKeyPoints	:	ITcVnContainer;	(* KeyPoints of the reference image, e.g. computed with F_VN_KeyPointsAndDescriptorsAKAZE (ContainerType_Vector_TcVnKeyPoint) *)
		ipRefDescriptors	:	ITcVnImage;	(* Descriptors of the reference image KeyPoints, e.g. computed with F_VN_KeyPointsAndDescriptorsAKAZE *)
		nRefImageWidth	:	UDINT;	(* Width of the reference image in pixels *)
		nRefImageHeight	:	UDINT;	(* Height of the reference image in pixels *)
		ipEdgePoints	:	REFERENCE TO ITcVnContainer;	(* Returns a container with the 4 edge points of the reference image transformed into ipSrcImage coordinates (ContainerType_Vector_TcVnPoint2_REAL) *)
		fMaxDist	:	REAL;	(* Maximum allowed descriptor distance (-1 disables this filter criterion) *)
		fMaxKnnRatio	:	REAL;	(* Maximum allowed distance ratio between first and second best match ([0..1], -1 disables this filter criterion) *)
		hrPrev	:	HRESULT;	(* HRESULT indicating the result of previous operations (If SUCCEEDED(hrPrev) equals false, no operation is executed.) *)
	END_VAR
	VAR_OUTPUT
		aPerspectiveTransform	:	TcVnMatrix3x3_LREAL;	(* Returns the perspective transformation matrix, which transforms the reference points to the source points *)
		nNumberOfGoodMatches	:	UDINT;	(* Return the number of good matches *)
		nNumberOfInliers	:	UDINT;	(* Return the number of inlier matches *)
	END_VAR

END_FUNCTION

// Functions/Keypoint Features/F_VN_KeyPointsAndDescriptorsAKAZE

	{attribute 'TcIecLibraryType'}
	{attribute 'external_name' := 'F_VN_KeyPointsAndDescriptorsAKAZE_GUID_AC11F1B8_F425_D686_8658_2A3527A9CAE7'}
	(* Detects keypoints and compute descriptors using the AKAZE method. *)
	FUNCTION F_VN_KeyPointsAndDescriptorsAKAZE : HRESULT
	VAR_INPUT
		ipSrcImage	:	ITcVnImage;	(* Source image *)
		ipKeyPoints	:	REFERENCE TO ITcVnContainer;	(* Returns a container which is filled with the keypoints (ContainerType_Vector_TcVnKeyPoint; Non-zero interface pointers are reused.) *)
		ipDescriptors	:	REFERENCE TO ITcVnImage;	(* Descriptor image (set to 0 if not required; 1 descriptor in each row; An appropriate image will be created if required.) *)
		hrPrev	:	HRESULT;	(* HRESULT indicating the result of previous operations (If SUCCEEDED(hrPrev) equals false, no operation is executed.) *)
	END_VAR

END_FUNCTION

// Functions/Keypoint Features/F_VN_FindReferenceKeyPointsInImageAKAZEExp

	{attribute 'TcIecLibraryType'}
	{attribute 'external_name' := 'F_VN_FindReferenceKeyPointsInImageAKAZEExp_GUID_C5CDBC97_9F14_DE21_AD79_676C896720A1'}
	(* Searches a reference image, represented by its AKAZE keypoints and corresponding descriptors, in a given source image. (expert function) *)
	FUNCTION F_VN_FindReferenceKeyPointsInImageAKAZEExp : HRESULT
	VAR_INPUT
		ipSrcImage	:	ITcVnImage;	(* Source image *)
		ipRefKeyPoints	:	ITcVnContainer;	(* KeyPoints of the reference image, e.g. computed with F_VN_KeyPointsAndDescriptorsAKAZE (ContainerType_Vector_TcVnKeyPoint) *)
		ipRefDescriptors	:	ITcVnImage;	(* Descriptors of the reference image KeyPoints, e.g. computed with F_VN_KeyPointsAndDescriptorsAKAZE *)
		nRefImageWidth	:	UDINT;	(* Width of the reference image in pixels *)
		nRefImageHeight	:	UDINT;	(* Height of the reference image in pixels *)
		ipEdgePoints	:	REFERENCE TO ITcVnContainer;	(* Returns a container with the 4 edge points of the reference image transformed into ipSrcImage coordinates (ContainerType_Vector_TcVnPoint2_REAL) *)
		fMaxDist	:	REAL;	(* Maximum allowed descriptor distance (-1 disables this filter criterion) *)
		fMaxKnnRatio	:	REAL;	(* Maximum allowed distance ratio between first and second best match ([0..1], -1 disables this filter criterion) *)
		eNormType	:	ETcVnNormalizationType;	(* Normalization type used for descriptor matching *)
		ipSrcImageMask	:	ITcVnImage;	(* Mask to specify, where to look for keypoints in ipSrcImage (set to 0 if no mask required) *)
	END_VAR
	VAR_IN_OUT
		stAkazeParams	:	TcVnParamsAKAZE;	(* Parameters to configure the keypoint and descriptor computation for ipSrcImage (resulting descriptors must be compatible to ipRefDescriptors!) *)
	END_VAR
	VAR_INPUT
		eAlgorithm	:	ETcVnEstimationAlgorithm;	(* Estimation algorithm used for computing the perspective transformation between the two point sets *)
		fReprojThreshold	:	LREAL;	(* Maximum allowed reprojection error to treat a point pair as an inlier (only used if eAlgorithm is RANSAC, RHO) *)
		nMaxIterations	:	UDINT;	(* Maximum number of RANSAC iterations *)
		fConfidence	:	LREAL;	(* Confidence (0..1) *)
		hrPrev	:	HRESULT;	(* HRESULT indicating the result of previous operations (If SUCCEEDED(hrPrev) equals false, no operation is executed.) *)
	END_VAR
	VAR_OUTPUT
		aPerspectiveTransform	:	TcVnMatrix3x3_LREAL;	(* Returns the perspective transformation matrix, which transforms the reference points to the source points  *)
		nNumberOfGoodMatches	:	UDINT;	(* Return the number of good matches *)
		nNumberOfInliers	:	UDINT;	(* Return the number of inlier matches *)
	END_VAR

END_FUNCTION

// Functions/Keypoint Features/F_VN_FindReferenceKeyPointsInImageBRISK

	{attribute 'TcIecLibraryType'}
	{attribute 'external_name' := 'F_VN_FindReferenceKeyPointsInImageBRISK_GUID_59596BB8_CDF7_DA8C_8704_693C28AB60AB'}
	(* Searches a reference image, represented by its BRISK keypoints and corresponding descriptors, in a given source image (uses the default TcVnParamsBRISK parameters). *)
	FUNCTION F_VN_FindReferenceKeyPointsInImageBRISK : HRESULT
	VAR_INPUT
		ipSrcImage	:	ITcVnImage;	(* Source image *)
		ipRefKeyPoints	:	ITcVnContainer;	(* KeyPoints of the reference image, e.g. computed with F_VN_KeyPointsAndDescriptorsBRISK (ContainerType_Vector_TcVnKeyPoint) *)
		ipRefDescriptors	:	ITcVnImage;	(* Descriptors of the reference image KeyPoints, e.g. computed with F_VN_KeyPointsAndDescriptorsBRISK *)
		nRefImageWidth	:	UDINT;	(* Width of the reference image in pixels *)
		nRefImageHeight	:	UDINT;	(* Height of the reference image in pixels *)
		ipEdgePoints	:	REFERENCE TO ITcVnContainer;	(* Returns a container with the 4 edge points of the reference image transformed into ipSrcImage coordinates (ContainerType_Vector_TcVnPoint2_REAL) *)
		fMaxDist	:	REAL;	(* Maximum allowed descriptor distance (-1 disables this filter criterion) *)
		fMaxKnnRatio	:	REAL;	(* Maximum allowed distance ratio between first and second best match ([0..1], -1 disables this filter criterion) *)
		hrPrev	:	HRESULT;	(* HRESULT indicating the result of previous operations (If SUCCEEDED(hrPrev) equals false, no operation is executed.) *)
	END_VAR
	VAR_OUTPUT
		aPerspectiveTransform	:	TcVnMatrix3x3_LREAL;	(* Returns the perspective transformation matrix, which transforms the reference points to the source points  *)
		nNumberOfGoodMatches	:	UDINT;	(* Return the number of good matches *)
		nNumberOfInliers	:	UDINT;	(* Return the number of inlier matches *)
	END_VAR

END_FUNCTION

// Functions/Keypoint Features/F_VN_KeyPointsAndDescriptorsBRISK

	{attribute 'TcIecLibraryType'}
	{attribute 'external_name' := 'F_VN_KeyPointsAndDescriptorsBRISK_GUID_1B2DB734_51EB_D0D4_B64D_A96941FF19E7'}
	(* Detects keypoints and compute descriptors using the BRISK method. *)
	FUNCTION F_VN_KeyPointsAndDescriptorsBRISK : HRESULT
	VAR_INPUT
		ipSrcImage	:	ITcVnImage;	(* Source image *)
		ipKeyPoints	:	REFERENCE TO ITcVnContainer;	(* Returns a container which is filled with the keypoints (ContainerType_Vector_TcVnKeyPoint; Non-zero interface pointers are reused.) *)
		ipDescriptors	:	REFERENCE TO ITcVnImage;	(* Descriptor image (set to 0 if not required; 1 descriptor in each row; An appropriate image will be created if required.) *)
		hrPrev	:	HRESULT;	(* HRESULT indicating the result of previous operations (If SUCCEEDED(hrPrev) equals false, no operation is executed.) *)
	END_VAR

END_FUNCTION

// Functions/Keypoint Features/F_VN_FindReferenceKeyPointsInImageBRISKExp

	{attribute 'TcIecLibraryType'}
	{attribute 'external_name' := 'F_VN_FindReferenceKeyPointsInImageBRISKExp_GUID_1B55C6DA_8589_DE50_AAD0_42730CD451F8'}
	(* Searches a reference image, represented by its BRISK keypoints and corresponding descriptors, in a given source image. (expert function) *)
	FUNCTION F_VN_FindReferenceKeyPointsInImageBRISKExp : HRESULT
	VAR_INPUT
		ipSrcImage	:	ITcVnImage;	(* Source image *)
		ipRefKeyPoints	:	ITcVnContainer;	(* KeyPoints of the reference image, e.g. computed with F_VN_KeyPointsAndDescriptorsBRISK (ContainerType_Vector_TcVnKeyPoint) *)
		ipRefDescriptors	:	ITcVnImage;	(* Descriptors of the reference image KeyPoints, e.g. computed with F_VN_KeyPointsAndDescriptorsBRISK *)
		nRefImageWidth	:	UDINT;	(* Width of the reference image in pixels *)
		nRefImageHeight	:	UDINT;	(* Height of the reference image in pixels *)
		ipEdgePoints	:	REFERENCE TO ITcVnContainer;	(* Returns a container with the 4 edge points of the reference image transformed into ipSrcImage coordinates (ContainerType_Vector_TcVnPoint2_REAL) *)
		fMaxDist	:	REAL;	(* Maximum allowed descriptor distance (-1 disables this filter criterion) *)
		fMaxKnnRatio	:	REAL;	(* Maximum allowed distance ratio between first and second best match ([0..1], -1 disables this filter criterion) *)
		eNormType	:	ETcVnNormalizationType;	(* Normalization type used for descriptor matching *)
		ipSrcImageMask	:	ITcVnImage;	(* Mask to specify, where to look for keypoints in ipSrcImage (set to 0 if no mask required) *)
	END_VAR
	VAR_IN_OUT
		stBriskParams	:	TcVnParamsBRISK;	(* Parameters to configure the keypoint and descriptor computation for ipSrcImage (resulting descriptors must be compatible to ipRefDescriptors!) *)
	END_VAR
	VAR_INPUT
		eAlgorithm	:	ETcVnEstimationAlgorithm;	(* Estimation algorithm used for computing the perspective transformation between the two point sets *)
		fReprojThreshold	:	LREAL;	(* Maximum allowed reprojection error to treat a point pair as an inlier (only used if eAlgorithm is RANSAC, RHO) *)
		nMaxIterations	:	UDINT;	(* Maximum number of RANSAC iterations *)
		fConfidence	:	LREAL;	(* Confidence (0..1) *)
		hrPrev	:	HRESULT;	(* HRESULT indicating the result of previous operations (If SUCCEEDED(hrPrev) equals false, no operation is executed.) *)
	END_VAR
	VAR_OUTPUT
		aPerspectiveTransform	:	TcVnMatrix3x3_LREAL;	(* Returns the perspective transformation matrix, which transforms the reference points to the source points  *)
		nNumberOfGoodMatches	:	UDINT;	(* Return the number of good matches *)
		nNumberOfInliers	:	UDINT;	(* Return the number of inlier matches *)
	END_VAR

END_FUNCTION

// Functions/Keypoint Features/F_VN_FindReferenceKeyPointsInImageORB

	{attribute 'TcIecLibraryType'}
	{attribute 'external_name' := 'F_VN_FindReferenceKeyPointsInImageORB_GUID_3818B428_FEB2_D432_8031_7955861D0617'}
	(* Searches a reference image, represented by its ORB keypoints and corresponding descriptors, in a given source image (uses the default TcVnParamsORB parameters). *)
	FUNCTION F_VN_FindReferenceKeyPointsInImageORB : HRESULT
	VAR_INPUT
		ipSrcImage	:	ITcVnImage;	(* Source image *)
		ipRefKeyPoints	:	ITcVnContainer;	(* KeyPoints of the reference image, e.g. computed with F_VN_KeyPointsAndDescriptorsORB (ContainerType_Vector_TcVnKeyPoint) *)
		ipRefDescriptors	:	ITcVnImage;	(* Descriptors of the reference image KeyPoints, e.g. computed with F_VN_KeyPointsAndDescriptorsORB *)
		nRefImageWidth	:	UDINT;	(* Width of the reference image in pixels *)
		nRefImageHeight	:	UDINT;	(* Height of the reference image in pixels *)
		ipEdgePoints	:	REFERENCE TO ITcVnContainer;	(* Returns a container with the 4 edge points of the reference image transformed into ipSrcImage coordinates (ContainerType_Vector_TcVnPoint2_REAL) *)
		fMaxDist	:	REAL;	(* Maximum allowed descriptor distance (-1 disables this filter criterion) *)
		fMaxKnnRatio	:	REAL;	(* Maximum allowed distance ratio between first and second best match ([0..1], -1 disables this filter criterion) *)
		hrPrev	:	HRESULT;	(* HRESULT indicating the result of previous operations (If SUCCEEDED(hrPrev) equals false, no operation is executed.) *)
	END_VAR
	VAR_OUTPUT
		aPerspectiveTransform	:	TcVnMatrix3x3_LREAL;	(* Returns the perspective transformation matrix, which transforms the reference points to the source points  *)
		nNumberOfGoodMatches	:	UDINT;	(* Return the number of good matches *)
		nNumberOfInliers	:	UDINT;	(* Return the number of inlier matches *)
	END_VAR

END_FUNCTION

// Functions/Keypoint Features/F_VN_KeyPointsAndDescriptorsORB

	{attribute 'TcIecLibraryType'}
	{attribute 'external_name' := 'F_VN_KeyPointsAndDescriptorsORB_GUID_00BBE309_9FDF_D1B3_B65F_8B3B201D9A3F'}
	(* Detects keypoints and compute descriptors using the ORB method. *)
	FUNCTION F_VN_KeyPointsAndDescriptorsORB : HRESULT
	VAR_INPUT
		ipSrcImage	:	ITcVnImage;	(* Source image *)
		ipKeyPoints	:	REFERENCE TO ITcVnContainer;	(* Returns a container which is filled with the keypoints (ContainerType_Vector_TcVnKeyPoint; Non-zero interface pointers are reused.) *)
		ipDescriptors	:	REFERENCE TO ITcVnImage;	(* Descriptor image (set to 0 if not required; 1 descriptor in each row; An appropriate image will be created if required.) *)
		hrPrev	:	HRESULT;	(* HRESULT indicating the result of previous operations (If SUCCEEDED(hrPrev) equals false, no operation is executed.) *)
	END_VAR

END_FUNCTION

// Functions/Keypoint Features/F_VN_FindReferenceKeyPointsInImageORBExp

	{attribute 'TcIecLibraryType'}
	{attribute 'external_name' := 'F_VN_FindReferenceKeyPointsInImageORBExp_GUID_E51C1141_A4AE_DE53_839A_65443B7981F6'}
	(* Searches a reference image, represented by its ORB keypoints and corresponding descriptors, in a given source image. (expert function) *)
	FUNCTION F_VN_FindReferenceKeyPointsInImageORBExp : HRESULT
	VAR_INPUT
		ipSrcImage	:	ITcVnImage;	(* Source image *)
		ipRefKeyPoints	:	ITcVnContainer;	(* KeyPoints of the reference image, e.g. computed with F_VN_KeyPointsAndDescriptorsORB (ContainerType_Vector_TcVnKeyPoint) *)
		ipRefDescriptors	:	ITcVnImage;	(* Descriptors of the reference image KeyPoints, e.g. computed with F_VN_KeyPointsAndDescriptorsORB *)
		nRefImageWidth	:	UDINT;	(* Width of the reference image in pixels *)
		nRefImageHeight	:	UDINT;	(* Height of the reference image in pixels *)
		ipEdgePoints	:	REFERENCE TO ITcVnContainer;	(* Returns a container with the 4 edge points of the reference image transformed into ipSrcImage coordinates (ContainerType_Vector_TcVnPoint2_REAL) *)
		fMaxDist	:	REAL;	(* Maximum allowed descriptor distance (-1 disables this filter criterion) *)
		fMaxKnnRatio	:	REAL;	(* Maximum allowed distance ratio between first and second best match ([0..1], -1 disables this filter criterion) *)
		eNormType	:	ETcVnNormalizationType;	(* Normalization type used for descriptor matching (HAMMING recommended for ORB, HAMMING2 if the ORB nBriefPoints parameter is 3 or 4) *)
		ipSrcImageMask	:	ITcVnImage;	(* Mask to specify, where to look for keypoints in ipSrcImage (set to 0 if no mask required) *)
	END_VAR
	VAR_IN_OUT
		stOrbParams	:	TcVnParamsORB;	(* Parameters to configure the keypoint and descriptor computation for ipSrcImage (resulting descriptors must be compatible to ipRefDescriptors!) *)
	END_VAR
	VAR_INPUT
		eAlgorithm	:	ETcVnEstimationAlgorithm;	(* Estimation algorithm used for computing the perspective transformation between the two point sets *)
		fReprojThreshold	:	LREAL;	(* Maximum allowed reprojection error to treat a point pair as an inlier (only used if eAlgorithm is RANSAC, RHO) *)
		nMaxIterations	:	UDINT;	(* Maximum number of RANSAC iterations *)
		fConfidence	:	LREAL;	(* Confidence (0..1) *)
		hrPrev	:	HRESULT;	(* HRESULT indicating the result of previous operations (If SUCCEEDED(hrPrev) equals false, no operation is executed.) *)
	END_VAR
	VAR_OUTPUT
		aPerspectiveTransform	:	TcVnMatrix3x3_LREAL;	(* Returns the perspective transformation matrix, which transforms the reference points to the source points  *)
		nNumberOfGoodMatches	:	UDINT;	(* Return the number of good matches *)
		nNumberOfInliers	:	UDINT;	(* Return the number of inlier matches *)
	END_VAR

END_FUNCTION

// Functions/Keypoint Features/F_VN_GetMatchCoordinates

	{attribute 'TcIecLibraryType'}
	{attribute 'external_name' := 'F_VN_GetMatchCoordinates_GUID_57611CBE_ACC8_D97E_8CEB_635BA370910C'}
	(* Return the coordinates of keypoints that match each other. *)
	FUNCTION F_VN_GetMatchCoordinates : HRESULT
	VAR_INPUT
		ipQueryKeyPoints	:	ITcVnContainer;	(* Container with query Keypoints (i.e. keypoints of a reference/template image) of type CTcVnContainer_Vector_TcVnKeyPoint *)
		ipTrainKeyPoints	:	ITcVnContainer;	(* Container with training Keypoints (i.e. keypoints of a source/input image) of type CTcVnContainer_Vector_TcVnKeyPoint *)
		ipMatches	:	ITcVnContainer;	(* Container with matches between query and train Keypoints (CTcVnContainer_Vector_TcVnDMatch). *)
		ipQueryCoordinates	:	REFERENCE TO ITcVnContainer;	(* Returns a container with the coordinates of keypoints from the query Keypoints that exist in ipMatches (CTcVnContainer_Vector_TcVnPoint2_REAL) *)
		ipTrainCoordinates	:	REFERENCE TO ITcVnContainer;	(* Returns a container with the coordinates of keypoints from the training Keypoints that exist in ipMatches (CTcVnContainer_Vector_TcVnPoint2_REAL) *)
		hrPrev	:	HRESULT;	(* HRESULT indicating the result of previous operations (If SUCCEEDED(hrPrev) equals false, no operation is executed.) *)
	END_VAR

END_FUNCTION

// Functions/Keypoint Features/F_VN_KeyPointsAGAST

	{attribute 'TcIecLibraryType'}
	{attribute 'external_name' := 'F_VN_KeyPointsAGAST_GUID_14F0C300_8C70_D5BC_B743_C03010F70BD5'}
	(* Detects keypoints using the AGAST method. *)
	FUNCTION F_VN_KeyPointsAGAST : HRESULT
	VAR_INPUT
		ipSrcImage	:	ITcVnImage;	(* Source image *)
		ipKeyPoints	:	REFERENCE TO ITcVnContainer;	(* Returns a container which is filled with the keypoints (ContainerType_Vector_TcVnKeyPoint; Non-zero interface pointers are reused.) *)
		hrPrev	:	HRESULT;	(* HRESULT indicating the result of previous operations (If SUCCEEDED(hrPrev) equals false, no operation is executed.) *)
	END_VAR

END_FUNCTION

// Functions/Keypoint Features/F_VN_KeyPointsAGASTExp

	{attribute 'TcIecLibraryType'}
	{attribute 'external_name' := 'F_VN_KeyPointsAGASTExp_GUID_038A822D_03B9_D397_8D7C_4DA9E4CDAFBA'}
	(* Detects keypoints using the AGAST method. (expert function) *)
	FUNCTION F_VN_KeyPointsAGASTExp : HRESULT
	VAR_INPUT
		ipSrcImage	:	ITcVnImage;	(* Source image *)
		ipKeyPoints	:	REFERENCE TO ITcVnContainer;	(* Returns a container which is filled with the keypoints (ContainerType_Vector_TcVnKeyPoint; Non-zero interface pointers are reused.) *)
		ipMask	:	ITcVnImage;	(* Mask to specify, where to look for keypoints (set to 0 if no mask required) *)
	END_VAR
	VAR_IN_OUT
		stParams	:	TcVnParamsAGAST;	(* Additional expert parameters *)
	END_VAR
	VAR_INPUT
		hrPrev	:	HRESULT;	(* HRESULT indicating the result of previous operations (If SUCCEEDED(hrPrev) equals false, no operation is executed.) *)
	END_VAR

END_FUNCTION

// Functions/Keypoint Features/F_VN_KeyPointsAndDescriptorsAKAZEExp

	{attribute 'TcIecLibraryType'}
	{attribute 'external_name' := 'F_VN_KeyPointsAndDescriptorsAKAZEExp_GUID_F41B3740_8046_DCD5_BADC_401EFA5D85EB'}
	(* Detects keypoints and compute descriptors using the AKAZE method. (expert function) *)
	FUNCTION F_VN_KeyPointsAndDescriptorsAKAZEExp : HRESULT
	VAR_INPUT
		ipSrcImage	:	ITcVnImage;	(* Source image *)
		ipKeyPoints	:	REFERENCE TO ITcVnContainer;	(* Returns a container which is filled with the keypoints (ContainerType_Vector_TcVnKeyPoint; Non-zero interface pointers are reused.) *)
		ipDescriptors	:	REFERENCE TO ITcVnImage;	(* Descriptor image (set to 0 if not required; 1 descriptor in each row; An appropriate image will be created if required.) *)
		ipMask	:	ITcVnImage;	(* Mask to specify, where to look for keypoints (set to 0 if no mask required) *)
	END_VAR
	VAR_IN_OUT
		stParams	:	TcVnParamsAKAZE;	(* Additional expert parameters *)
	END_VAR
	VAR_INPUT
		hrPrev	:	HRESULT;	(* HRESULT indicating the result of previous operations (If SUCCEEDED(hrPrev) equals false, no operation is executed.) *)
	END_VAR

END_FUNCTION

// Functions/Keypoint Features/F_VN_KeyPointsAndDescriptorsBRISKExp

	{attribute 'TcIecLibraryType'}
	{attribute 'external_name' := 'F_VN_KeyPointsAndDescriptorsBRISKExp_GUID_4580C7F5_33D6_D729_9822_40B96B9F4567'}
	(* Detects keypoints and compute descriptors using the BRISK method. (expert function) *)
	FUNCTION F_VN_KeyPointsAndDescriptorsBRISKExp : HRESULT
	VAR_INPUT
		ipSrcImage	:	ITcVnImage;	(* Source image *)
		ipKeyPoints	:	REFERENCE TO ITcVnContainer;	(* Returns a container which is filled with the keypoints (ContainerType_Vector_TcVnKeyPoint; Non-zero interface pointers are reused.) *)
		ipDescriptors	:	REFERENCE TO ITcVnImage;	(* Descriptor image (set to 0 if not required; 1 descriptor in each row; An appropriate image will be created if required.) *)
		ipMask	:	ITcVnImage;	(* Mask to specify, where to look for keypoints (set to 0 if no mask required) *)
	END_VAR
	VAR_IN_OUT
		stParams	:	TcVnParamsBRISK;	(* Additional expert parameters *)
	END_VAR
	VAR_INPUT
		hrPrev	:	HRESULT;	(* HRESULT indicating the result of previous operations (If SUCCEEDED(hrPrev) equals false, no operation is executed.) *)
	END_VAR

END_FUNCTION

// Functions/Keypoint Features/F_VN_KeyPointsAndDescriptorsKAZE

	{attribute 'TcIecLibraryType'}
	{attribute 'external_name' := 'F_VN_KeyPointsAndDescriptorsKAZE_GUID_54933517_5CAA_DA2C_8550_07B3DE85C197'}
	(* Detects keypoints and compute descriptors using the KAZE method. *)
	FUNCTION F_VN_KeyPointsAndDescriptorsKAZE : HRESULT
	VAR_INPUT
		ipSrcImage	:	ITcVnImage;	(* Source image *)
		ipKeyPoints	:	REFERENCE TO ITcVnContainer;	(* Returns a container which is filled with the keypoints (ContainerType_Vector_TcVnKeyPoint; Non-zero interface pointers are reused.) *)
		ipDescriptors	:	REFERENCE TO ITcVnImage;	(* Descriptor image (set to 0 if not required; 1 descriptor in each row; An appropriate image will be created if required.) *)
		hrPrev	:	HRESULT;	(* HRESULT indicating the result of previous operations (If SUCCEEDED(hrPrev) equals false, no operation is executed.) *)
	END_VAR

END_FUNCTION

// Functions/Keypoint Features/F_VN_KeyPointsAndDescriptorsKAZEExp

	{attribute 'TcIecLibraryType'}
	{attribute 'external_name' := 'F_VN_KeyPointsAndDescriptorsKAZEExp_GUID_34206243_3A30_D64F_96FE_473198C68457'}
	(* Detects keypoints and compute descriptors using the KAZE method. (expert function) *)
	FUNCTION F_VN_KeyPointsAndDescriptorsKAZEExp : HRESULT
	VAR_INPUT
		ipSrcImage	:	ITcVnImage;	(* Source image *)
		ipKeyPoints	:	REFERENCE TO ITcVnContainer;	(* Returns a container which is filled with the keypoints (ContainerType_Vector_TcVnKeyPoint; Non-zero interface pointers are reused.) *)
		ipDescriptors	:	REFERENCE TO ITcVnImage;	(* Descriptor image (set to 0 if not required; 1 descriptor in each row; An appropriate image will be created if required.) *)
		ipMask	:	ITcVnImage;	(* Mask to specify, where to look for keypoints (set to 0 if no mask required) *)
	END_VAR
	VAR_IN_OUT
		stParams	:	TcVnParamsKAZE;	(* Additional expert parameters *)
	END_VAR
	VAR_INPUT
		hrPrev	:	HRESULT;	(* HRESULT indicating the result of previous operations (If SUCCEEDED(hrPrev) equals false, no operation is executed.) *)
	END_VAR

END_FUNCTION

// Functions/Keypoint Features/F_VN_KeyPointsAndDescriptorsORBExp

	{attribute 'TcIecLibraryType'}
	{attribute 'external_name' := 'F_VN_KeyPointsAndDescriptorsORBExp_GUID_7D231AB1_EA2F_D9A1_977A_29F2BA282107'}
	(* Detect keypoints and compute descriptors using the ORB method. (expert function) *)
	FUNCTION F_VN_KeyPointsAndDescriptorsORBExp : HRESULT
	VAR_INPUT
		ipSrcImage	:	ITcVnImage;	(* Source image *)
		ipKeyPoints	:	REFERENCE TO ITcVnContainer;	(* Returns a container which is filled with the keypoints (ContainerType_Vector_TcVnKeyPoint; Non-zero interface pointers are reused.) *)
		ipDescriptors	:	REFERENCE TO ITcVnImage;	(* Descriptor image (set to 0 if not required; 1 descriptor in each row; An appropriate image will be created if required.) *)
		ipMask	:	ITcVnImage;	(* Mask to specify, where to look for keypoints (set to 0 if no mask required) *)
	END_VAR
	VAR_IN_OUT
		stParams	:	TcVnParamsORB;	(* Additional expert parameters *)
	END_VAR
	VAR_INPUT
		hrPrev	:	HRESULT;	(* HRESULT indicating the result of previous operations (If SUCCEEDED(hrPrev) equals false, no operation is executed.) *)
	END_VAR

END_FUNCTION

// Functions/Keypoint Features/F_VN_KeyPointsFAST

	{attribute 'TcIecLibraryType'}
	{attribute 'external_name' := 'F_VN_KeyPointsFAST_GUID_CC2B8A02_7781_D93B_BFFA_E3E51A2C9BCB'}
	(* Detects keypoints using the FAST method. *)
	FUNCTION F_VN_KeyPointsFAST : HRESULT
	VAR_INPUT
		ipSrcImage	:	ITcVnImage;	(* Source image (single-channel). *)
		ipKeyPoints	:	REFERENCE TO ITcVnContainer;	(* Returns a container which is filled with the keypoints (ContainerType_Vector_TcVnKeyPoint; Non-zero interface pointers are reused.) *)
		hrPrev	:	HRESULT;	(* HRESULT indicating the result of previous operations (If SUCCEEDED(hrPrev) equals false, no operation is executed.) *)
	END_VAR

END_FUNCTION

// Functions/Keypoint Features/F_VN_KeyPointsFASTExp

	{attribute 'TcIecLibraryType'}
	{attribute 'external_name' := 'F_VN_KeyPointsFASTExp_GUID_16F12969_61CB_DE8F_A036_8F154D52BA3E'}
	(* Detects keypoints using the FAST method. (expert function) *)
	FUNCTION F_VN_KeyPointsFASTExp : HRESULT
	VAR_INPUT
		ipSrcImage	:	ITcVnImage;	(* Source image *)
		ipKeyPoints	:	REFERENCE TO ITcVnContainer;	(* Returns a container which is filled with the keypoints (ContainerType_Vector_TcVnKeyPoint; Non-zero interface pointers are reused.) *)
		ipMask	:	ITcVnImage;	(* Mask to specify, where to look for keypoints (set to 0 if no mask required) *)
	END_VAR
	VAR_IN_OUT
		stParams	:	TcVnParamsFAST;	(* Additional expert parameters *)
	END_VAR
	VAR_INPUT
		hrPrev	:	HRESULT;	(* HRESULT indicating the result of previous operations (If SUCCEEDED(hrPrev) equals false, no operation is executed.) *)
	END_VAR

END_FUNCTION

// Functions/Keypoint Features/F_VN_KeyPointsGFTT

	{attribute 'TcIecLibraryType'}
	{attribute 'external_name' := 'F_VN_KeyPointsGFTT_GUID_D4AE6E9C_E008_DC58_816A_F7E9C9F8CD4F'}
	(* Detects keypoints using the GFTT method, which detects strong corners. *)
	FUNCTION F_VN_KeyPointsGFTT : HRESULT
	VAR_INPUT
		ipSrcImage	:	ITcVnImage;	(* Source image *)
		ipKeyPoints	:	REFERENCE TO ITcVnContainer;	(* Returns a container which is filled with the keypoints (ContainerType_Vector_TcVnKeyPoint; Non-zero interface pointers are reused.) *)
		hrPrev	:	HRESULT;	(* HRESULT indicating the result of previous operations (If SUCCEEDED(hrPrev) equals false, no operation is executed.) *)
	END_VAR

END_FUNCTION

// Functions/Keypoint Features/F_VN_KeyPointsGFTTExp

	{attribute 'TcIecLibraryType'}
	{attribute 'external_name' := 'F_VN_KeyPointsGFTTExp_GUID_58D07B54_13D6_DEB2_99C5_8F00E8B3120E'}
	(* Detects keypoints using the GFTT method, which detects strong corners. (expert function) *)
	FUNCTION F_VN_KeyPointsGFTTExp : HRESULT
	VAR_INPUT
		ipSrcImage	:	ITcVnImage;	(* Source image *)
		ipKeyPoints	:	REFERENCE TO ITcVnContainer;	(* Returns a container which is filled with the keypoints (ContainerType_Vector_TcVnKeyPoint; Non-zero interface pointers are reused.) *)
		ipMask	:	ITcVnImage;	(* Mask to specify, where to look for keypoints (set to 0 if no mask required) *)
	END_VAR
	VAR_IN_OUT
		stParams	:	TcVnParamsGFTT;	(* Additional expert parameters *)
	END_VAR
	VAR_INPUT
		hrPrev	:	HRESULT;	(* HRESULT indicating the result of previous operations (If SUCCEEDED(hrPrev) equals false, no operation is executed.) *)
	END_VAR

END_FUNCTION

// Functions/Keypoint Features/F_VN_KeyPointsMSER

	{attribute 'TcIecLibraryType'}
	{attribute 'external_name' := 'F_VN_KeyPointsMSER_GUID_AA88890D_70BC_D4C9_899C_14B84ADB97D8'}
	(* Detects keypoints using the MSER method. *)
	FUNCTION F_VN_KeyPointsMSER : HRESULT
	VAR_INPUT
		ipSrcImage	:	ITcVnImage;	(* Source image *)
		ipKeyPoints	:	REFERENCE TO ITcVnContainer;	(* Returns a container which is filled with the keypoints (ContainerType_Vector_TcVnKeyPoint; Non-zero interface pointers are reused.) *)
		hrPrev	:	HRESULT;	(* HRESULT indicating the result of previous operations (If SUCCEEDED(hrPrev) equals false, no operation is executed.) *)
	END_VAR

END_FUNCTION

// Functions/Keypoint Features/F_VN_KeyPointsMSERExp

	{attribute 'TcIecLibraryType'}
	{attribute 'external_name' := 'F_VN_KeyPointsMSERExp_GUID_5857DB59_C2E5_DBC3_B0F9_A479A73BC7F1'}
	(* Detects keypoints using the MSER method. (expert function) *)
	FUNCTION F_VN_KeyPointsMSERExp : HRESULT
	VAR_INPUT
		ipSrcImage	:	ITcVnImage;	(* Source image *)
		ipKeyPoints	:	REFERENCE TO ITcVnContainer;	(* Returns a container which is filled with the keypoints (ContainerType_Vector_TcVnKeyPoint; Non-zero interface pointers are reused.) *)
		ipMask	:	ITcVnImage;	(* Mask to specify, where to look for keypoints (set to 0 if no mask required) *)
	END_VAR
	VAR_IN_OUT
		stParams	:	TcVnParamsMSER;	(* Additional expert parameters *)
	END_VAR
	VAR_INPUT
		hrPrev	:	HRESULT;	(* HRESULT indicating the result of previous operations (If SUCCEEDED(hrPrev) equals false, no operation is executed.) *)
	END_VAR

END_FUNCTION

// Functions/Keypoint Features/F_VN_KeyPointsSB

	{attribute 'TcIecLibraryType'}
	{attribute 'external_name' := 'F_VN_KeyPointsSB_GUID_D9453E80_D8CB_D3C1_A98F_A2D1AFE0CB38'}
	(* Detects keypoints using a Simple Blob method
          - several iterations apply different thresholds to source image
          - connected components (blobs) are detected
          - the center and radius of the blobs are returned as keypoints *)
	FUNCTION F_VN_KeyPointsSB : HRESULT
	VAR_INPUT
		ipSrcImage	:	ITcVnImage;	(* Source image *)
		ipKeyPoints	:	REFERENCE TO ITcVnContainer;	(* Returns a container which is filled with the keypoints (ContainerType_Vector_TcVnKeyPoint; Non-zero interface pointers are reused.) *)
		hrPrev	:	HRESULT;	(* HRESULT indicating the result of previous operations (If SUCCEEDED(hrPrev) equals false, no operation is executed.) *)
	END_VAR

END_FUNCTION

// Functions/Keypoint Features/F_VN_KeyPointsSBExp

	{attribute 'TcIecLibraryType'}
	{attribute 'external_name' := 'F_VN_KeyPointsSBExp_GUID_724188B6_31E1_DAF0_BE8E_6840ABEAA1EB'}
	(* Detects keypoints using a Simple Blob method (expert function)
          - several iterations apply different thresholds to source image
          - connected components (blobs) are detected
          - the center and radius of the blobs are returned as keypoints *)
	FUNCTION F_VN_KeyPointsSBExp : HRESULT
	VAR_INPUT
		ipSrcImage	:	ITcVnImage;	(* Source image *)
		ipKeyPoints	:	REFERENCE TO ITcVnContainer;	(* Returns a container which is filled with the keypoints (ContainerType_Vector_TcVnKeyPoint; Non-zero interface pointers are reused.) *)
		ipMask	:	ITcVnImage;	(* Mask to specify, where to look for keypoints (optional, set to 0 if not required) *)
	END_VAR
	VAR_IN_OUT
		stParams	:	TcVnParamsSB;	(* Several parameters to filter the detected blobs *)
	END_VAR
	VAR_INPUT
		hrPrev	:	HRESULT;	(* HRESULT indicating the result of previous operations (If SUCCEEDED(hrPrev) equals false, no operation is executed.) *)
	END_VAR

END_FUNCTION

// Functions/Keypoint Features/F_VN_MatchDescriptorsBF

	{attribute 'TcIecLibraryType'}
	{attribute 'external_name' := 'F_VN_MatchDescriptorsBF_GUID_402396C2_483B_DA31_A52B_1D67B5F820C4'}
	(* Match descriptors using a brute force approach. *)
	FUNCTION F_VN_MatchDescriptorsBF : HRESULT
	VAR_INPUT
		ipQueryDescriptors	:	ITcVnImage;	(* Query descriptors (i.e. descriptors of a reference/template image) *)
		ipTrainDescriptors	:	ITcVnImage;	(* Training descriptors (i.e. descriptors of a source/input image) *)
		ipMatches	:	REFERENCE TO ITcVnContainer;	(* Returns a container which is filled with the descriptor matches (ContainerType_Vector_TcVnDMatch; Non-zero interface pointers are reused.) *)
		hrPrev	:	HRESULT;	(* HRESULT indicating the result of previous operations (If SUCCEEDED(hrPrev) equals false, no operation is executed.) *)
	END_VAR

END_FUNCTION

// Functions/Keypoint Features/F_VN_MatchDescriptorsBFExp

	{attribute 'TcIecLibraryType'}
	{attribute 'external_name' := 'F_VN_MatchDescriptorsBFExp_GUID_B136CDA3_CC74_D098_9E88_253C80D3DCD8'}
	(* Match descriptors using a brute force approach. (expert function) *)
	FUNCTION F_VN_MatchDescriptorsBFExp : HRESULT
	VAR_INPUT
		ipQueryDescriptors	:	ITcVnImage;	(* Query descriptors (i.e. descriptors of a reference/template image) *)
		ipTrainDescriptors	:	ITcVnImage;	(* Training descriptors (i.e. descriptors of a source/input image) *)
		ipMatches	:	REFERENCE TO ITcVnContainer;	(* Returns a container which is filled with the descriptor matches (ContainerType_Vector_TcVnDMatch; Non-zero interface pointers are reused.) *)
		ipMask	:	ITcVnImage;	(* Mask to specify permissable matches, i.e. query[i] can be matched with train[j] only if mask[i][j] != 0 (set to 0 if no mask required) *)
		eNormType	:	ETcVnNormalizationType;	(* Normalization type (only L1, L2, L2SQR, HAMMING, HAMMING2 supported). HAMMING2 should be used for ORB descriptors if the ORB nBriefPoints parameter is 3 or 4) *)
		bCrossCheck	:	BOOL;	(* If true, only consistent matches are returned, i.e. query->train and train->query detect the same match *)
		hrPrev	:	HRESULT;	(* HRESULT indicating the result of previous operations (If SUCCEEDED(hrPrev) equals false, no operation is executed.) *)
	END_VAR

END_FUNCTION

// Functions/Keypoint Features/F_VN_MatchDescriptorsFlannLsh

	{attribute 'TcIecLibraryType'}
	{attribute 'external_name' := 'F_VN_MatchDescriptorsFlannLsh_GUID_99BD9580_4E33_D219_8585_6923F2EB02AA'}
	(* Match descriptors using a FLANN based approach with LSH index. *)
	FUNCTION F_VN_MatchDescriptorsFlannLsh : HRESULT
	VAR_INPUT
		ipQueryDescriptors	:	ITcVnImage;	(* Query descriptors (i.e. descriptors of a reference/template image) *)
		ipTrainDescriptors	:	ITcVnImage;	(* Training descriptors (i.e. descriptors of a source/input image) *)
		ipMatches	:	REFERENCE TO ITcVnContainer;	(* Returns a container which is filled with the descriptor matches (ContainerType_Vector_TcVnDMatch; Non-zero interface pointers are reused.) *)
		hrPrev	:	HRESULT;	(* HRESULT indicating the result of previous operations (If SUCCEEDED(hrPrev) equals false, no operation is executed.) *)
	END_VAR

END_FUNCTION

// Functions/Keypoint Features/F_VN_MatchDescriptorsFlannLshExp

	{attribute 'TcIecLibraryType'}
	{attribute 'external_name' := 'F_VN_MatchDescriptorsFlannLshExp_GUID_550199C5_ADA9_D3F4_9262_02F0460E0C21'}
	(* Match descriptors using a FLANN based approach with LSH index. (expert function) *)
	FUNCTION F_VN_MatchDescriptorsFlannLshExp : HRESULT
	VAR_INPUT
		ipQueryDescriptors	:	ITcVnImage;	(* Query descriptors (i.e. descriptors of a reference/template image) *)
		ipTrainDescriptors	:	ITcVnImage;	(* Training descriptors (i.e. descriptors of a source/input image) *)
		ipMatches	:	REFERENCE TO ITcVnContainer;	(* Returns a container which is filled with the descriptor matches (ContainerType_Vector_TcVnDMatch; Non-zero interface pointers are reused.) *)
		nTableNumber	:	UDINT;	(* Number of tables *)
		nKeySize	:	UDINT;	(* Key size *)
		nMultiProbeLevel	:	UDINT;	(* Multi-probe level *)
		nChecks	:	UDINT;	(* Maximum number of visited leafs when searching for neighbors *)
		hrPrev	:	HRESULT;	(* HRESULT indicating the result of previous operations (If SUCCEEDED(hrPrev) equals false, no operation is executed.) *)
	END_VAR

END_FUNCTION

// Functions/Keypoint Features/F_VN_MatchDescriptorsKnnBF

	{attribute 'TcIecLibraryType'}
	{attribute 'external_name' := 'F_VN_MatchDescriptorsKnnBF_GUID_F09DB3A2_580C_DD8F_ADC0_3DAF92ACB540'}
	(* Match descriptors (k nearest neighbors) using a brute force approach. *)
	FUNCTION F_VN_MatchDescriptorsKnnBF : HRESULT
	VAR_INPUT
		ipQueryDescriptors	:	ITcVnImage;	(* Query descriptors (i.e. descriptors of a reference/template image) *)
		ipTrainDescriptors	:	ITcVnImage;	(* Training descriptors (i.e. descriptors of a source/input image) *)
		ipMatches	:	REFERENCE TO ITcVnContainer;	(* Returns a container which is filled with the descriptor matches (ContainerType_Vector_Vector_TcVnDMatch; Non-zero interface pointers are reused.) *)
		nK	:	UDINT;	(* Number of required best train matches for each query descriptor (i.e. nk := 2) *)
		hrPrev	:	HRESULT;	(* HRESULT indicating the result of previous operations (If SUCCEEDED(hrPrev) equals false, no operation is executed.) *)
	END_VAR

END_FUNCTION

// Functions/Keypoint Features/F_VN_MatchDescriptorsKnnBFExp

	{attribute 'TcIecLibraryType'}
	{attribute 'external_name' := 'F_VN_MatchDescriptorsKnnBFExp_GUID_BCEAB2D6_BEFA_D68F_9553_84B4A5138454'}
	(* Match descriptors (k nearest neighbors) using a brute force approach. (expert function) *)
	FUNCTION F_VN_MatchDescriptorsKnnBFExp : HRESULT
	VAR_INPUT
		ipQueryDescriptors	:	ITcVnImage;	(* Query descriptors (i.e. descriptors of a reference/template image) *)
		ipTrainDescriptors	:	ITcVnImage;	(* Training descriptors (i.e. descriptors of a source/input image) *)
		ipMatches	:	REFERENCE TO ITcVnContainer;	(* Returns a container which is filled with the descriptor matches (ContainerType_Vector_Vector_TcVnDMatch; Non-zero interface pointers are reused.) *)
		nK	:	UDINT;	(* Number of required best train matches for each query descriptor (i.e. nk := 2) *)
		ipMask	:	ITcVnImage;	(* Mask to specify permissable matches, i.e. query[i] can be matched with train[j] only if mask[i][j] != 0 (set to 0 if no mask required) *)
		bCompactResult	:	BOOL;	(* If true, matches vector does not contain entries for fully masked-out query descriptors *)
		eNormType	:	ETcVnNormalizationType;	(* Normalization type (only L1, L2, L2SQR, HAMMING, HAMMING2 supported). HAMMING2 should be used for ORB descriptors if the ORB nBriefPoints parameter is 3 or 4) *)
		bCrossCheck	:	BOOL;	(* If true, only consistent matches are returned, i.e. query->train and train->query detect the same match (only used if nK = 1) *)
		hrPrev	:	HRESULT;	(* HRESULT indicating the result of previous operations (If SUCCEEDED(hrPrev) equals false, no operation is executed.) *)
	END_VAR

END_FUNCTION

// Functions/Keypoint Features/F_VN_MatchDescriptorsKnnFlannLsh

	{attribute 'TcIecLibraryType'}
	{attribute 'external_name' := 'F_VN_MatchDescriptorsKnnFlannLsh_GUID_3B91B730_37F0_DDFE_A3E9_0D3CE74D4BCF'}
	(* Match descriptors (k nearest neighbors) using a FLANN based approach with LSH index. *)
	FUNCTION F_VN_MatchDescriptorsKnnFlannLsh : HRESULT
	VAR_INPUT
		ipQueryDescriptors	:	ITcVnImage;	(* Query descriptors (i.e. descriptors of a reference/template image) *)
		ipTrainDescriptors	:	ITcVnImage;	(* Training descriptors (i.e. descriptors of a source/input image) *)
		ipMatches	:	REFERENCE TO ITcVnContainer;	(* Returns a container which is filled with the descriptor matches (ContainerType_Vector_Vector_TcVnDMatch; Non-zero interface pointers are reused.) *)
		nK	:	UDINT;	(* Number of required best train matches for each query descriptor (i.e. nk := 2) *)
		hrPrev	:	HRESULT;	(* HRESULT indicating the result of previous operations (If SUCCEEDED(hrPrev) equals false, no operation is executed.) *)
	END_VAR

END_FUNCTION

// Functions/Keypoint Features/F_VN_MatchDescriptorsKnnFlannLshExp

	{attribute 'TcIecLibraryType'}
	{attribute 'external_name' := 'F_VN_MatchDescriptorsKnnFlannLshExp_GUID_3729EF0B_7C72_DD9F_BEBD_186067719D97'}
	(* Match descriptors (k nearest neighbors) using a FLANN based approach with LSH index. (expert function) *)
	FUNCTION F_VN_MatchDescriptorsKnnFlannLshExp : HRESULT
	VAR_INPUT
		ipQueryDescriptors	:	ITcVnImage;	(* Query descriptors (i.e. descriptors of a reference/template image) *)
		ipTrainDescriptors	:	ITcVnImage;	(* Training descriptors (i.e. descriptors of a source/input image) *)
		ipMatches	:	REFERENCE TO ITcVnContainer;	(* Returns a container which is filled with the descriptor matches (ContainerType_Vector_Vector_TcVnDMatch; Non-zero interface pointers are reused.) *)
		nK	:	UDINT;	(* Number of required best train matches for each query descriptor (i.e. nk := 2) *)
		nTableNumber	:	UDINT;	(* Number of tables *)
		nKeySize	:	UDINT;	(* Key size *)
		nMultiProbeLevel	:	UDINT;	(* Multi-probe level *)
		nChecks	:	UDINT;	(* Maximum number of visited leafs when searching for neighbors *)
		hrPrev	:	HRESULT;	(* HRESULT indicating the result of previous operations (If SUCCEEDED(hrPrev) equals false, no operation is executed.) *)
	END_VAR

END_FUNCTION

// Functions/Keypoint Features/F_VN_RegionsMSER

	{attribute 'TcIecLibraryType'}
	{attribute 'external_name' := 'F_VN_RegionsMSER_GUID_A6C1EA01_03ED_DDBE_BA76_DD65E3500C40'}
	(* Detects regions using the MSER method. *)
	FUNCTION F_VN_RegionsMSER : HRESULT
	VAR_INPUT
		ipSrcImage	:	ITcVnImage;	(* Source image *)
		ipRegions	:	REFERENCE TO ITcVnContainer;	(* Returns a container which is filled with the region points (ContainerType_Vector_Vector_TcVnPoint2_DINT; Non-zero interface pointers are reused.) *)
		ipBoundingBoxes	:	REFERENCE TO ITcVnContainer;	(* Returns a container which is filled with the region bounding boxes (ContainerType_Vector_TcVnRectangle_DINT; Non-zero interface pointers are reused.) *)
		hrPrev	:	HRESULT;	(* HRESULT indicating the result of previous operations (If SUCCEEDED(hrPrev) equals false, no operation is executed.) *)
	END_VAR

END_FUNCTION

// Functions/Keypoint Features/F_VN_RegionsMSERExp

	{attribute 'TcIecLibraryType'}
	{attribute 'external_name' := 'F_VN_RegionsMSERExp_GUID_173D8FB4_D472_D362_9B54_A46EC147CD37'}
	(* Detects regions using the MSER method. (expert function) *)
	FUNCTION F_VN_RegionsMSERExp : HRESULT
	VAR_INPUT
		ipSrcImage	:	ITcVnImage;	(* Source image *)
		ipRegions	:	REFERENCE TO ITcVnContainer;	(* Returns a container which is filled with the region points (ContainerType_Vector_Vector_TcVnPoint2_DINT; Non-zero interface pointers are reused.) *)
		ipBoundingBoxes	:	REFERENCE TO ITcVnContainer;	(* Returns a container which is filled with the region bounding boxes (ContainerType_Vector_TcVnRectangle_DINT; Non-zero interface pointers are reused.) *)
	END_VAR
	VAR_IN_OUT
		stParams	:	TcVnParamsMSER;	(* Additional expert parameters *)
	END_VAR
	VAR_INPUT
		hrPrev	:	HRESULT;	(* HRESULT indicating the result of previous operations (If SUCCEEDED(hrPrev) equals false, no operation is executed.) *)
	END_VAR

END_FUNCTION

// Functions/Code Quality/F_VN_GradeBarcode

	{attribute 'TcIecLibraryType'}
	{attribute 'external_name' := 'F_VN_GradeBarcode_GUID_8A51F6A8_1DFE_D77C_A653_AC6007D8E53C'}
	(* Grades a 1D barcode according to ISO / IEC 15416:2016. Requires uniform illumination, good focus and the image sensor plane parallel to the code plane to achieve meaningful results. *)
	FUNCTION F_VN_GradeBarcode : HRESULT
	VAR_INPUT
		ipSrcImage	:	ITcVnImage;	(* Source image, only containing the horizontally aligned barcode region (USINT, 1 channel, including quiet zones on left and right, excluding Text or empty space on more than 10% total height on top or bottom) *)
		ipDecodedData	:	REFERENCE TO ITcVnContainer;	(* Returns the decoded data (ContainerType_String_SINT) *)
	END_VAR
	VAR_IN_OUT
		stCodeGrades	:	TcVnCodeGrades1D;	(* Returns the code grades in the range from 0 (very bad) to 4 (very good) *)
	END_VAR
	VAR_INPUT
		eBarcodeType	:	ETcVnBarcodeType;	(* Type of the barcode (supported: CODE39, CODE128, EAN8, EAN13, ITF, UPCA, UPCE) *)
		hrPrev	:	HRESULT;	(* HRESULT indicating the result of previous operations (If SUCCEEDED(hrPrev) equals false, no operation is executed.) *)
	END_VAR
	VAR_OUTPUT
		fAngleDeg	:	REAL;	(* Returns the approximate clockwise rotation angle in degree *)
	END_VAR

END_FUNCTION

// Functions/Code Quality/F_VN_GradeBarcodeExp

	{attribute 'TcIecLibraryType'}
	{attribute 'external_name' := 'F_VN_GradeBarcodeExp_GUID_0380B83D_84AF_D95C_AB18_5EE5EFDC72D6'}
	(* Grades a 1D barcode according to ISO / IEC 15416:2016. Requires uniform illumination, good focus and the image sensor plane parallel to the code plane to achieve meaningful results. (expert function) *)
	FUNCTION F_VN_GradeBarcodeExp : HRESULT
	VAR_INPUT
		ipSrcImage	:	ITcVnImage;	(* Source image, only containing the horizontally aligned barcode region (USINT, 1 channel, including quiet zones on left and right, excluding Text or empty space on more than 10% total height on top or bottom) *)
		ipDecodedData	:	REFERENCE TO ITcVnContainer;	(* Returns the decoded data (ContainerType_String_SINT) *)
	END_VAR
	VAR_IN_OUT
		stCodeGrades	:	TcVnCodeGrades1D;	(* Returns the code grades in the range from 0 (very bad) to 4 (very good) *)
	END_VAR
	VAR_INPUT
		eBarcodeType	:	ETcVnBarcodeType;	(* Type of the barcode (supported: CODE39, CODE128, EAN8, EAN13, ITF, UPCA, UPCE) *)
		eSearchDirection	:	ETcVnBarcodeSearchDirection;	(* Barcode search direction (BSD_ANY first tries horizontal, then vertical) *)
		ipResultVisualization	:	REFERENCE TO ITcVnImage;	(* Returns a visualization of the scan lines (optional, set to 0 if not required). Grades are color coded: >= 3 as green, >= 2 as light blue, >= 1 as orange, < 1 as red *)
		ipScanLineInfo	:	REFERENCE TO ITcVnContainer;	(* Returns additional scan line info for further evaluation, e.g. to use PlotIntensityProfile for visualization (optional, set to 0 if not required; ContainerType_Vector_TcVnVector3_REAL, containing [row index, overall grade, threshold]) *)
		ipContour	:	REFERENCE TO ITcVnContainer;	(* Returns the 4 approximate code corner points, including the quiet zone (optional, set to 0 if not required; ContainerType_Vector_TcVnPoint2_DINT) *)
		hrPrev	:	HRESULT;	(* HRESULT indicating the result of previous operations (If SUCCEEDED(hrPrev) equals false, no operation is executed.) *)
	END_VAR
	VAR_OUTPUT
		fAngleDeg	:	REAL;	(* Returns the approximate clockwise rotation angle in degree *)
	END_VAR

END_FUNCTION

// Functions/Code Quality/F_VN_GradeDataMatrixCode

	{attribute 'TcIecLibraryType'}
	{attribute 'external_name' := 'F_VN_GradeDataMatrixCode_GUID_ABD6460D_FD7B_D40A_A9CD_D5A5338D3790'}
	(* Grades a Data Matrix code (ECC200) according to ISO / IEC 15415:2011. Requires uniform illumination, good focus and the image sensor plane parallel to the code plane to achieve meaningful results. *)
	FUNCTION F_VN_GradeDataMatrixCode : HRESULT
	VAR_INPUT
		ipSrcImage	:	ITcVnImage;	(* Source image, only containing the Data Matrix code region (USINT, 1 channel, including quiet zone) *)
		ipDecodedData	:	REFERENCE TO ITcVnContainer;	(* Returns the decoded data (ContainerType_String_SINT) *)
	END_VAR
	VAR_IN_OUT
		stCodeGrades	:	TcVnCodeGradesDM;	(* Returns the code grades in the range from 0 (very bad) to 4 (very good) *)
	END_VAR
	VAR_INPUT
		fModuleWidth	:	REAL;	(* Minimum module width of the code in the image (in pixels). Must be at least 3, preferably 5 - 8. *)
		hrPrev	:	HRESULT;	(* HRESULT indicating the result of previous operations (If SUCCEEDED(hrPrev) equals false, no operation is executed.) *)
	END_VAR
	VAR_OUTPUT
		fAngleDeg	:	REAL;	(* Returns the clockwise rotation angle in degree *)
	END_VAR

END_FUNCTION

// Functions/Code Quality/F_VN_GradeDataMatrixCodeExp

